LIN {X 0,Y 226.3,Z 547.719,A -85,B 0,C 180,E1 -21646.905,E2 -21646.905} C_VEL
LIN {X 0,Y 219.819,Z 558.471,A -85,B 0,C 180,E1 -21649.654,E2 -21649.654} C_VEL
LIN {X 0,Y 214.009,Z 567.653,A -85,B 0,C 180,E1 -21652.59,E2 -21652.59} C_VEL
LIN {X 0,Y 207.988,Z 576.689,A -85,B 0,C 180,E1 -21656.115,E2 -21656.115} C_VEL
LIN {X 0,Y 202.319,Z 585.085,A -85,B 0,C 180,E1 -21660.276,E2 -21660.276} C_VEL
LIN {X 0,Y 197.664,Z 592.031,A -85,B 0,C 180,E1 -21664.745,E2 -21664.745} C_VEL
LIN {X 0,Y 193.918,Z 597.973,A -85,B 0,C 180,E1 -21669.862,E2 -21669.862} C_VEL
LIN {X 0,Y 192.297,Z 600.784,A -85,B 0,C 180,E1 -21673,E2 -21673} C_VEL
LIN {X 0,Y 190.826,Z 603.573,A -85,B 0,C 180,E1 -21677.234,E2 -21677.234} C_VEL
LIN {X 0,Y 190.2,Z 605.482,A -85,B 0,C 180,E1 -21681.501,E2 -21681.501} C_VEL
LIN {X 0,Y 190.122,Z 606.399,A -85,B 0,C 180,E1 -21686.441,E2 -21686.441} C_VEL
LIN {X 0,Y 190.28,Z 606.307,A -85,B 0,C 180,E1 -21690.001,E2 -21690.001} C_VEL
LIN {X 0,Y 190.16,Z 605.178,A -85,B 0,C 180,E1 -21694.24,E2 -21694.24} C_VEL
LIN {X 0,Y 190.208,Z 603.116,A -85,B 0,C 180,E1 -21698.5,E2 -21698.5} C_VEL
LIN {X 0,Y 190.815,Z 599.908,A -85,B 0,C 180,E1 -21702.768,E2 -21702.768} C_VEL
LIN {X 0,Y 192.236,Z 595.672,A -85,B 0,C 180,E1 -21707.007,E2 -21707.007} C_VEL
LIN {X 0,Y 194.259,Z 590.216,A -85,B 0,C 180,E1 -21711.21,E2 -21711.21} C_VEL
LIN {X 0,Y 197.197,Z 583.475,A -85,B 0,C 180,E1 -21715.32,E2 -21715.32} C_VEL
LIN {X 0,Y 200.967,Z 575.348,A -85,B 0,C 180,E1 -21719.314,E2 -21719.314} C_VEL
LIN {X 0,Y 205.672,Z 565.618,A -85,B 0,C 180,E1 -21723.143,E2 -21723.143} C_VEL
LIN {X 0,Y 209.744,Z 557.011,A -85,B 0,C 180,E1 -21725.901,E2 -21725.901} C_VEL
LIN {X 0,Y 215.012,Z 545.421,A -85,B 0,C 180,E1 -21728.992,E2 -21728.992} C_VEL
LIN {X 0,Y 220.42,Z 532.769,A -85,B 0,C 180,E1 -21731.728,E2 -21731.728} C_VEL
LIN {X 0,Y 225.253,Z 520.818,A -85,B 0,C 180,E1 -21733.809,E2 -21733.809} C_VEL
LIN {X 0,Y 230.337,Z 506.753,A -85,B 0,C 180,E1 -21735.81,E2 -21735.81} C_VEL
LIN {X 0,Y 234.904,Z 492.399,A -85,B 0,C 180,E1 -21737.455,E2 -21737.455} C_VEL
LIN {X 0,Y 239.123,Z 476.927,A -85,B 0,C 180,E1 -21738.863,E2 -21738.863} C_VEL
LIN {X 0,Y 242.624,Z 461.116,A -85,B 0,C 180,E1 -21739.978,E2 -21739.978} C_VEL
LIN {X 0,Y 245.67,Z 444.06,A -85,B 0,C 180,E1 -21740.823,E2 -21740.823} C_VEL
LIN {X 0,Y 247.577,Z 427.936,A -85,B 0,C 180,E1 -21741.39,E2 -21741.39} C_VEL
LIN {X 0,Y 254.979,Z 326.261,A -85,B 0,C 180,E1 -21744.097,E2 -21744.097} C_VEL
LIN {X 0,Y 248.761,Z 313.085,A -85,B 0,C 180,E1 -21746.361,E2 -21746.361} C_VEL
LIN {X 0,Y 242.88,Z 301.521,A -85,B 0,C 180,E1 -21748.649,E2 -21748.649} C_VEL
LIN {X 0,Y 237.783,Z 292.318,A -85,B 0,C 180,E1 -21750.757,E2 -21750.757} C_VEL
LIN {X 0,Y 234.658,Z 287.086,A -85,B 0,C 180,E1 -21752.117,E2 -21752.117} C_VEL
LIN {X 0,Y 228.084,Z 277.705,A -85,B 0,C 180,E1 -21755.145,E2 -21755.145} C_VEL
LIN {X 0,Y 222.612,Z 270.114,A -85,B 0,C 180,E1 -21757.951,E2 -21757.951} C_VEL
LIN {X 0,Y 219.484,Z 266.04,A -85,B 0,C 180,E1 -21759.698,E2 -21759.698} C_VEL
LIN {X 0,Y 216.41,Z 261.942,A -85,B 0,C 180,E1 -21761.562,E2 -21761.562} C_VEL
LIN {X 0,Y 212.892,Z 257.748,A -85,B 0,C 180,E1 -21763.827,E2 -21763.827} C_VEL
LIN {X 0,Y 211.789,Z 256.222,A -85,B 0,C 180,E1 -21764.605,E2 -21764.605} C_VEL
LIN {X 0,Y 209.031,Z 253.204,A -85,B 0,C 180,E1 -21766.625,E2 -21766.625} C_VEL
LIN {X 0,Y 207.994,Z 251.231,A -85,B 0,C 180,E1 -21767.53,E2 -21767.53} C_VEL
LIN {X 0,Y 205.278,Z 248.973,A -85,B 0,C 180,E1 -21769.744,E2 -21769.744} C_VEL
LIN {X 0,Y 203.429,Z 245.607,A -85,B 0,C 180,E1 -21771.605,E2 -21771.605} C_VEL
LIN {X 0,Y 200.503,Z 243.62,A -85,B 0,C 180,E1 -21774.595,E2 -21774.595} C_VEL
LIN {X 0,Y 198.935,Z 241.093,A -85,B 0,C 180,E1 -21776.646,E2 -21776.646} C_VEL
LIN {X 0,Y 198.424,Z 239.663,A -85,B 0,C 180,E1 -21777.462,E2 -21777.462} C_VEL
LIN {X 0,Y 194.087,Z 236.776,A -85,B 0,C 180,E1 -21785.194,E2 -21785.194} C_VEL
LIN {X 0,Y 193.073,Z 234.315,A -85,B 0,C 180,E1 -21790.001,E2 -21790.001} C_VEL
LIN {X 0,Y 192.86,Z 234.123,A -85,B 0,C 180,E1 -21794.24,E2 -21794.24} C_VEL
LIN {X 0,Y 193.402,Z 236.089,A -85,B 0,C 180,E1 -21799.09,E2 -21799.09} C_VEL
LIN {X 0,Y 196.596,Z 239.298,A -85,B 0,C 180,E1 -21806.543,E2 -21806.543} C_VEL
LIN {X 0,Y 198.274,Z 240.054,A -85,B 0,C 180,E1 -21808.935,E2 -21808.935} C_VEL
LIN {X 0,Y 199.346,Z 242.603,A -85,B 0,C 180,E1 -21810.597,E2 -21810.597} C_VEL
LIN {X 0,Y 201.756,Z 245.019,A -85,B 0,C 180,E1 -21813.336,E2 -21813.336} C_VEL
LIN {X 0,Y 203.301,Z 246.022,A -85,B 0,C 180,E1 -21814.85,E2 -21814.85} C_VEL
LIN {X 0,Y 204.976,Z 248.974,A -85,B 0,C 180,E1 -21816.565,E2 -21816.565} C_VEL
LIN {X 0,Y 207.674,Z 251.22,A -85,B 0,C 180,E1 -21818.769,E2 -21818.769} C_VEL
LIN {X 0,Y 210.371,Z 255.153,A -85,B 0,C 180,E1 -21820.945,E2 -21820.945} C_VEL
LIN {X 0,Y 212.372,Z 257.041,A -85,B 0,C 180,E1 -21822.332,E2 -21822.332} C_VEL
LIN {X 0,Y 215.023,Z 260.684,A -85,B 0,C 180,E1 -21824.12,E2 -21824.12} C_VEL
LIN {X 0,Y 216.456,Z 262.166,A -85,B 0,C 180,E1 -21825.008,E2 -21825.008} C_VEL
LIN {X 0,Y 219.505,Z 266.13,A -85,B 0,C 180,E1 -21826.844,E2 -21826.844} C_VEL
LIN {X 0,Y 224.279,Z 272.472,A -85,B 0,C 180,E1 -21829.46,E2 -21829.46} C_VEL
LIN {X 0,Y 230.144,Z 280.518,A -85,B 0,C 180,E1 -21832.356,E2 -21832.356} C_VEL
LIN {X 0,Y 237.496,Z 291.276,A -85,B 0,C 180,E1 -21835.609,E2 -21835.609} C_VEL
LIN {X 0,Y 246.014,Z 305.014,A -85,B 0,C 180,E1 -21838.984,E2 -21838.984} C_VEL
LIN {X 0,Y 252.643,Z 316.674,A -85,B 0,C 180,E1 -21841.37,E2 -21841.37} C_VEL
LIN {X 0,Y 255.065,Z 321.147,A -85,B 0,C 180,E1 -21842.207,E2 -21842.207} C_VEL
LIN {X 0,Y 247.736,Z 420.872,A -85,B 0,C 180,E1 -21844.872,E2 -21844.872} C_VEL
LIN {X 0,Y 245.585,Z 437.685,A -85,B 0,C 180,E1 -21845.54,E2 -21845.54} C_VEL
LIN {X 0,Y 242.828,Z 453.469,A -85,B 0,C 180,E1 -21846.436,E2 -21846.436} C_VEL
LIN {X 0,Y 239.503,Z 468.656,A -85,B 0,C 180,E1 -21847.575,E2 -21847.575} C_VEL
LIN {X 0,Y 235.477,Z 483.687,A -85,B 0,C 180,E1 -21849.013,E2 -21849.013} C_VEL
LIN {X 0,Y 230.919,Z 498.153,A -85,B 0,C 180,E1 -21850.751,E2 -21850.751} C_VEL
LIN {X 0,Y 226.04,Z 511.98,A -85,B 0,C 180,E1 -21852.82,E2 -21852.82} C_VEL
LIN {X 0,Y 220.734,Z 525.239,A -85,B 0,C 180,E1 -21855.243,E2 -21855.243} C_VEL
LIN {X 0,Y 215.258,Z 537.956,A -85,B 0,C 180,E1 -21858.134,E2 -21858.134} C_VEL
LIN {X 0,Y 209.942,Z 549.371,A -85,B 0,C 180,E1 -21861.335,E2 -21861.335} C_VEL
LIN {X 0,Y 205.245,Z 559.035,A -85,B 0,C 180,E1 -21864.704,E2 -21864.704} C_VEL
LIN {X 0,Y 200.912,Z 567.881,A -85,B 0,C 180,E1 -21868.496,E2 -21868.496} C_VEL
LIN {X 0,Y 197.029,Z 575.994,A -85,B 0,C 180,E1 -21872.859,E2 -21872.859} C_VEL
LIN {X 0,Y 194.041,Z 582.465,A -85,B 0,C 180,E1 -21877.282,E2 -21877.282} C_VEL
LIN {X 0,Y 192.072,Z 587.326,A -85,B 0,C 180,E1 -21881.609,E2 -21881.609} C_VEL
LIN {X 0,Y 190.587,Z 591.369,A -85,B 0,C 180,E1 -21886.512,E2 -21886.512} C_VEL
LIN {X 0,Y 189.824,Z 594.152,A -85,B 0,C 180,E1 -21891.729,E2 -21891.729} C_VEL
LIN {X 0,Y 189.656,Z 595.421,A -85,B 0,C 180,E1 -21896.402,E2 -21896.402} C_VEL
LIN {X 0,Y 189.956,Z 595.502,A -85,B 0,C 180,E1 -21901.195,E2 -21901.195} C_VEL
LIN {X 0,Y 190.879,Z 594.328,A -85,B 0,C 180,E1 -21906.092,E2 -21906.092} C_VEL
LIN {X 0,Y 192.629,Z 591.858,A -85,B 0,C 180,E1 -21911.049,E2 -21911.049} C_VEL
LIN {X 0,Y 195.361,Z 587.97,A -85,B 0,C 180,E1 -21916.011,E2 -21916.011} C_VEL
LIN {X 0,Y 199.252,Z 582.546,A -85,B 0,C 180,E1 -21920.892,E2 -21920.892} C_VEL
LIN {X 0,Y 203.207,Z 577.04,A -85,B 0,C 180,E1 -21924.614,E2 -21924.614} C_VEL
LIN {X 0,Y 209.079,Z 568.863,A -85,B 0,C 180,E1 -21928.937,E2 -21928.937} C_VEL
LIN {X 0,Y 214.504,Z 561.069,A -85,B 0,C 180,E1 -21932.203,E2 -21932.203} C_VEL
LIN {X 0,Y 221.257,Z 550.841,A -85,B 0,C 180,E1 -21935.611,E2 -21935.611} C_VEL
LIN {X 0,Y 228.118,Z 539.48,A -85,B 0,C 180,E1 -21938.616,E2 -21938.616} C_VEL
LIN {X 0,Y 234.856,Z 527.408,A -85,B 0,C 180,E1 -21941.148,E2 -21941.148} C_VEL
LIN {X 0,Y 241.301,Z 514.567,A -85,B 0,C 180,E1 -21943.339,E2 -21943.339} C_VEL
LIN {X 0,Y 247.296,Z 501.19,A -85,B 0,C 180,E1 -21945.181,E2 -21945.181} C_VEL
LIN {X 0,Y 252.741,Z 487.284,A -85,B 0,C 180,E1 -21946.713,E2 -21946.713} C_VEL
LIN {X 0,Y 257.863,Z 471.68,A -85,B 0,C 180,E1 -21948.089,E2 -21948.089} C_VEL
LIN {X 0,Y 261.833,Z 457.05,A -85,B 0,C 180,E1 -21949.095,E2 -21949.095} C_VEL
LIN {X 0,Y 265.125,Z 441.997,A -85,B 0,C 180,E1 -21949.899,E2 -21949.899} C_VEL
LIN {X 0,Y 267.848,Z 425.319,A -85,B 0,C 180,E1 -21950.519,E2 -21950.519} C_VEL
LIN {X 0,Y 272.094,Z 380.522,A -85,B 0,C 180,E1 -21951.669,E2 -21951.669} C_VEL
LIN {X 0,Y 276.451,Z 332.828,A -85,B 0,C 180,E1 -21952.851,E2 -21952.851} C_VEL
LIN {X 0,Y 272.688,Z 325.115,A -85,B 0,C 180,E1 -21955.176,E2 -21955.176} C_VEL
LIN {X 0,Y 268.508,Z 317.322,A -85,B 0,C 180,E1 -21958.203,E2 -21958.203} C_VEL
LIN {X 0,Y 266.207,Z 313.483,A -85,B 0,C 180,E1 -21960.156,E2 -21960.156} C_VEL
LIN {X 0,Y 263.602,Z 308.901,A -85,B 0,C 180,E1 -21962.925,E2 -21962.925} C_VEL
LIN {X 0,Y 262.122,Z 306.157,A -85,B 0,C 180,E1 -21964.992,E2 -21964.992} C_VEL
LIN {X 0,Y 260.235,Z 303.911,A -85,B 0,C 180,E1 -21968.582,E2 -21968.582} C_VEL
LIN {X 0,Y 259.761,Z 301.619,A -85,B 0,C 180,E1 -21971.359,E2 -21971.359} C_VEL
LIN {X 0,Y 259.671,Z 301.612,A -85,B 0,C 180,E1 -21973.484,E2 -21973.484} C_VEL
LIN {X 0,Y 261.393,Z 305.792,A -85,B 0,C 180,E1 -21979.607,E2 -21979.607} C_VEL
LIN {X 0,Y 261.99,Z 306.539,A -85,B 0,C 180,E1 -21980.538,E2 -21980.538} C_VEL
LIN {X 0,Y 263.625,Z 309.473,A -85,B 0,C 180,E1 -21982.8,E2 -21982.8} C_VEL
LIN {X 0,Y 264.588,Z 311.792,A -85,B 0,C 180,E1 -21983.958,E2 -21983.958} C_VEL
LIN {X 0,Y 265.403,Z 315.135,A -85,B 0,C 180,E1 -21985.005,E2 -21985.005} C_VEL
LIN {X 0,Y 266.944,Z 323.106,A -85,B 0,C 180,E1 -21986.933,E2 -21986.933} C_VEL
LIN {X 0,Y 268.315,Z 328.069,A -85,B 0,C 180,E1 -21988.267,E2 -21988.267} C_VEL
LIN {X 0,Y 270.696,Z 333.766,A -85,B 0,C 180,E1 -21990.065,E2 -21990.065} C_VEL
LIN {X 0,Y 272.946,Z 339.745,A -85,B 0,C 180,E1 -21991.648,E2 -21991.648} C_VEL
LIN {X 0,Y 264.303,Z 430.241,A -85,B 0,C 180,E1 -21993.891,E2 -21993.891} C_VEL
LIN {X 0,Y 261.773,Z 445.91,A -85,B 0,C 180,E1 -21994.435,E2 -21994.435} C_VEL
LIN {X 0,Y 257.966,Z 462.562,A -85,B 0,C 180,E1 -21995.185,E2 -21995.185} C_VEL
LIN {X 0,Y 253.496,Z 478.126,A -85,B 0,C 180,E1 -21996.152,E2 -21996.152} C_VEL
LIN {X 0,Y 247.91,Z 494.137,A -85,B 0,C 180,E1 -21997.462,E2 -21997.462} C_VEL
LIN {X 0,Y 241.934,Z 508.77,A -85,B 0,C 180,E1 -21999.009,E2 -21999.009} C_VEL
LIN {X 0,Y 235.575,Z 522.278,A -85,B 0,C 180,E1 -22000.799,E2 -22000.799} C_VEL
LIN {X 0,Y 229.471,Z 533.923,A -85,B 0,C 180,E1 -22002.69,E2 -22002.69} C_VEL
LIN {X 0,Y 222.174,Z 546.633,A -85,B 0,C 180,E1 -22005.266,E2 -22005.266} C_VEL
LIN {X 0,Y 214.44,Z 558.899,A -85,B 0,C 180,E1 -22008.421,E2 -22008.421} C_VEL
LIN {X 0,Y 207.554,Z 569.21,A -85,B 0,C 180,E1 -22011.834,E2 -22011.834} C_VEL
LIN {X 0,Y 201.341,Z 577.918,A -85,B 0,C 180,E1 -22015.444,E2 -22015.444} C_VEL
LIN {X 0,Y 195.442,Z 586.085,A -85,B 0,C 180,E1 -22019.774,E2 -22019.774} C_VEL
LIN {X 0,Y 191.179,Z 592.098,A -85,B 0,C 180,E1 -22023.825,E2 -22023.825} C_VEL
LIN {X 0,Y 187.164,Z 597.975,A -85,B 0,C 180,E1 -22029.102,E2 -22029.102} C_VEL
LIN {X 0,Y 184.556,Z 602.217,A -85,B 0,C 180,E1 -22034.541,E2 -22034.541} C_VEL
LIN {X 0,Y 183.396,Z 604.501,A -85,B 0,C 180,E1 -22038.954,E2 -22038.954} C_VEL
LIN {X 0,Y 182.995,Z 605.853,A -85,B 0,C 180,E1 -22043.385,E2 -22043.385} C_VEL
LIN {X 0,Y 183.056,Z 606.213,A -85,B 0,C 180,E1 -22047.8,E2 -22047.8} C_VEL
LIN {X 0,Y 183.184,Z 606.069,A -85,B 0,C 180,E1 -22050.001,E2 -22050.001} C_VEL
LIN {X 0,Y 183.072,Z 604.899,A -85,B 0,C 180,E1 -22054.404,E2 -22054.404} C_VEL
LIN {X 0,Y 183.146,Z 602.78,A -85,B 0,C 180,E1 -22058.83,E2 -22058.83} C_VEL
LIN {X 0,Y 184.161,Z 598.607,A -85,B 0,C 180,E1 -22064.363,E2 -22064.363} C_VEL
LIN {X 0,Y 186.011,Z 593.473,A -85,B 0,C 180,E1 -22069.167,E2 -22069.167} C_VEL
LIN {X 0,Y 188.244,Z 588.146,A -85,B 0,C 180,E1 -22073.08,E2 -22073.08} C_VEL
LIN {X 0,Y 191.587,Z 581.058,A -85,B 0,C 180,E1 -22077.293,E2 -22077.293} C_VEL
LIN {X 0,Y 195.858,Z 572.422,A -85,B 0,C 180,E1 -22081.353,E2 -22081.353} C_VEL
LIN {X 0,Y 200.377,Z 563.506,A -85,B 0,C 180,E1 -22084.747,E2 -22084.747} C_VEL
LIN {X 0,Y 205.384,Z 553.105,A -85,B 0,C 180,E1 -22088.02,E2 -22088.02} C_VEL
LIN {X 0,Y 211.125,Z 540.871,A -85,B 0,C 180,E1 -22091.105,E2 -22091.105} C_VEL
LIN {X 0,Y 216.562,Z 528.481,A -85,B 0,C 180,E1 -22093.6,E2 -22093.6} C_VEL
LIN {X 0,Y 221.922,Z 514.889,A -85,B 0,C 180,E1 -22095.836,E2 -22095.836} C_VEL
LIN {X 0,Y 226.912,Z 500.869,A -85,B 0,C 180,E1 -22097.686,E2 -22097.686} C_VEL
LIN {X 0,Y 231.705,Z 485.342,A -85,B 0,C 180,E1 -22099.314,E2 -22099.314} C_VEL
LIN {X 0,Y 235.829,Z 469.309,A -85,B 0,C 180,E1 -22100.621,E2 -22100.621} C_VEL
LIN {X 0,Y 239.096,Z 453.413,A -85,B 0,C 180,E1 -22101.585,E2 -22101.585} C_VEL
LIN {X 0,Y 241.685,Z 437.265,A -85,B 0,C 180,E1 -22102.272,E2 -22102.272} C_VEL
LIN {X 0,Y 243.531,Z 417.107,A -85,B 0,C 180,E1 -22102.898,E2 -22102.898} C_VEL
LIN {X 0,Y 250.181,Z 328.977,A -85,B 0,C 180,E1 -22105.231,E2 -22105.231} C_VEL
LIN {X 0,Y 243.246,Z 314.287,A -85,B 0,C 180,E1 -22107.888,E2 -22107.888} C_VEL
LIN {X 0,Y 236.492,Z 301.128,A -85,B 0,C 180,E1 -22110.706,E2 -22110.706} C_VEL
LIN {X 0,Y 231.829,Z 292.97,A -85,B 0,C 180,E1 -22112.792,E2 -22112.792} C_VEL
LIN {X 0,Y 224.763,Z 282.709,A -85,B 0,C 180,E1 -22116.179,E2 -22116.179} C_VEL
LIN {X 0,Y 219.991,Z 276.007,A -85,B 0,C 180,E1 -22118.737,E2 -22118.737} C_VEL
LIN {X 0,Y 216.99,Z 272.049,A -85,B 0,C 180,E1 -22120.48,E2 -22120.48} C_VEL
LIN {X 0,Y 213.383,Z 267.331,A -85,B 0,C 180,E1 -22122.757,E2 -22122.757} C_VEL
LIN {X 0,Y 210.463,Z 263.477,A -85,B 0,C 180,E1 -22124.764,E2 -22124.764} C_VEL
LIN {X 0,Y 206.967,Z 259.331,A -85,B 0,C 180,E1 -22127.435,E2 -22127.435} C_VEL
LIN {X 0,Y 205.872,Z 257.674,A -85,B 0,C 180,E1 -22128.38,E2 -22128.38} C_VEL
LIN {X 0,Y 203.302,Z 255.168,A -85,B 0,C 180,E1 -22130.597,E2 -22130.597} C_VEL
LIN {X 0,Y 201.743,Z 252.369,A -85,B 0,C 180,E1 -22132.242,E2 -22132.242} C_VEL
LIN {X 0,Y 198.832,Z 250.084,A -85,B 0,C 180,E1 -22135.391,E2 -22135.391} C_VEL
LIN {X 0,Y 197.37,Z 247.437,A -85,B 0,C 180,E1 -22137.441,E2 -22137.441} C_VEL
LIN {X 0,Y 197.068,Z 246.554,A -85,B 0,C 180,E1 -22137.956,E2 -22137.956} C_VEL
LIN {X 0,Y 192.948,Z 243.573,A -85,B 0,C 180,E1 -22145.749,E2 -22145.749} C_VEL
LIN {X 0,Y 192.092,Z 241.306,A -85,B 0,C 180,E1 -22150.235,E2 -22150.235} C_VEL
LIN {X 0,Y 191.895,Z 241.115,A -85,B 0,C 180,E1 -22153.772,E2 -22153.772} C_VEL
LIN {X 0,Y 192.338,Z 242.935,A -85,B 0,C 180,E1 -22158.591,E2 -22158.591} C_VEL
LIN {X 0,Y 195.167,Z 246.109,A -85,B 0,C 180,E1 -22165.809,E2 -22165.809} C_VEL
LIN {X 0,Y 196.89,Z 246.955,A -85,B 0,C 180,E1 -22168.377,E2 -22168.377} C_VEL
LIN {X 0,Y 198.457,Z 250.027,A -85,B 0,C 180,E1 -22170.749,E2 -22170.749} C_VEL
LIN {X 0,Y 201.129,Z 252.313,A -85,B 0,C 180,E1 -22173.699,E2 -22173.699} C_VEL
LIN {X 0,Y 201.816,Z 253.005,A -85,B 0,C 180,E1 -22174.409,E2 -22174.409} C_VEL
LIN {X 0,Y 203.854,Z 256.203,A -85,B 0,C 180,E1 -22176.491,E2 -22176.491} C_VEL
LIN {X 0,Y 206.224,Z 258.311,A -85,B 0,C 180,E1 -22178.474,E2 -22178.474} C_VEL
LIN {X 0,Y 208.536,Z 261.69,A -85,B 0,C 180,E1 -22180.376,E2 -22180.376} C_VEL
LIN {X 0,Y 210.45,Z 263.668,A -85,B 0,C 180,E1 -22181.764,E2 -22181.764} C_VEL
LIN {X 0,Y 213.581,Z 267.699,A -85,B 0,C 180,E1 -22183.906,E2 -22183.906} C_VEL
LIN {X 0,Y 218.451,Z 274.056,A -85,B 0,C 180,E1 -22186.916,E2 -22186.916} C_VEL
LIN {X 0,Y 223.976,Z 281.525,A -85,B 0,C 180,E1 -22189.934,E2 -22189.934} C_VEL
LIN {X 0,Y 231.139,Z 291.963,A -85,B 0,C 180,E1 -22193.409,E2 -22193.409} C_VEL
LIN {X 0,Y 237.448,Z 301.854,A -85,B 0,C 180,E1 -22196.169,E2 -22196.169} C_VEL
LIN {X 0,Y 245.36,Z 315.183,A -85,B 0,C 180,E1 -22199.295,E2 -22199.295} C_VEL
LIN {X 0,Y 250.208,Z 324.114,A -85,B 0,C 180,E1 -22201.067,E2 -22201.067} C_VEL
LIN {X 0,Y 242.664,Z 422.976,A -85,B 0,C 180,E1 -22203.731,E2 -22203.731} C_VEL
LIN {X 0,Y 240.324,Z 440,A -85,B 0,C 180,E1 -22204.447,E2 -22204.447} C_VEL
LIN {X 0,Y 237.325,Z 455.867,A -85,B 0,C 180,E1 -22205.39,E2 -22205.39} C_VEL
LIN {X 0,Y 233.921,Z 470.539,A -85,B 0,C 180,E1 -22206.541,E2 -22206.541} C_VEL
LIN {X 0,Y 229.831,Z 485.302,A -85,B 0,C 180,E1 -22208.001,E2 -22208.001} C_VEL
LIN {X 0,Y 224.788,Z 500.514,A -85,B 0,C 180,E1 -22209.884,E2 -22209.884} C_VEL
LIN {X 0,Y 219.617,Z 514.379,A -85,B 0,C 180,E1 -22212.06,E2 -22212.06} C_VEL
LIN {X 0,Y 214.603,Z 526.286,A -85,B 0,C 180,E1 -22214.325,E2 -22214.325} C_VEL
LIN {X 0,Y 208.931,Z 538.914,A -85,B 0,C 180,E1 -22217.29,E2 -22217.29} C_VEL
LIN {X 0,Y 203.471,Z 550.176,A -85,B 0,C 180,E1 -22220.556,E2 -22220.556} C_VEL
LIN {X 0,Y 198.74,Z 559.505,A -85,B 0,C 180,E1 -22223.91,E2 -22223.91} C_VEL
LIN {X 0,Y 194.114,Z 568.532,A -85,B 0,C 180,E1 -22227.925,E2 -22227.925} C_VEL
LIN {X 0,Y 190.362,Z 576.056,A -85,B 0,C 180,E1 -22232.115,E2 -22232.115} C_VEL
LIN {X 0,Y 187.322,Z 582.298,A -85,B 0,C 180,E1 -22236.462,E2 -22236.462} C_VEL
LIN {X 0,Y 185.204,Z 587.21,A -85,B 0,C 180,E1 -22240.937,E2 -22240.937} C_VEL
LIN {X 0,Y 183.694,Z 591.029,A -85,B 0,C 180,E1 -22245.533,E2 -22245.533} C_VEL
LIN {X 0,Y 182.822,Z 593.775,A -85,B 0,C 180,E1 -22250.24,E2 -22250.24} C_VEL
LIN {X 0,Y 182.536,Z 595.332,A -85,B 0,C 180,E1 -22255.056,E2 -22255.056} C_VEL
LIN {X 0,Y 182.588,Z 595.725,A -85,B 0,C 180,E1 -22257.713,E2 -22257.713} C_VEL
LIN {X 0,Y 183.027,Z 595.601,A -85,B 0,C 180,E1 -22262.518,E2 -22262.518} C_VEL
LIN {X 0,Y 184.195,Z 594.221,A -85,B 0,C 180,E1 -22267.623,E2 -22267.623} C_VEL
LIN {X 0,Y 186.313,Z 591.474,A -85,B 0,C 180,E1 -22272.763,E2 -22272.763} C_VEL
LIN {X 0,Y 189.494,Z 587.299,A -85,B 0,C 180,E1 -22277.88,E2 -22277.88} C_VEL
LIN {X 0,Y 193.89,Z 581.559,A -85,B 0,C 180,E1 -22282.884,E2 -22282.884} C_VEL
LIN {X 0,Y 198.881,Z 575.19,A -85,B 0,C 180,E1 -22287.061,E2 -22287.061} C_VEL
LIN {X 0,Y 204.17,Z 568.171,A -85,B 0,C 180,E1 -22290.654,E2 -22290.654} C_VEL
LIN {X 0,Y 210.637,Z 559.222,A -85,B 0,C 180,E1 -22294.294,E2 -22294.294} C_VEL
LIN {X 0,Y 217.462,Z 549.157,A -85,B 0,C 180,E1 -22297.542,E2 -22297.542} C_VEL
LIN {X 0,Y 224.655,Z 537.774,A -85,B 0,C 180,E1 -22300.457,E2 -22300.457} C_VEL
LIN {X 0,Y 232.036,Z 524.859,A -85,B 0,C 180,E1 -22303.08,E2 -22303.08} C_VEL
LIN {X 0,Y 239.031,Z 510.982,A -85,B 0,C 180,E1 -22305.316,E2 -22305.316} C_VEL
LIN {X 0,Y 245.137,Z 497.106,A -85,B 0,C 180,E1 -22307.096,E2 -22307.096} C_VEL
LIN {X 0,Y 250.914,Z 482.098,A -85,B 0,C 180,E1 -22308.613,E2 -22308.613} C_VEL
LIN {X 0,Y 256.012,Z 466.15,A -85,B 0,C 180,E1 -22309.889,E2 -22309.889} C_VEL
LIN {X 0,Y 259.969,Z 450.749,A -85,B 0,C 180,E1 -22310.852,E2 -22310.852} C_VEL
LIN {X 0,Y 263.326,Z 433.993,A -85,B 0,C 180,E1 -22311.595,E2 -22311.595} C_VEL
LIN {X 0,Y 265.649,Z 416.43,A -85,B 0,C 180,E1 -22312.131,E2 -22312.131} C_VEL
LIN {X 0,Y 273.16,Z 336.704,A -85,B 0,C 180,E1 -22314.093,E2 -22314.093} C_VEL
LIN {X 0,Y 269.895,Z 329.796,A -85,B 0,C 180,E1 -22316.306,E2 -22316.306} C_VEL
LIN {X 0,Y 266.062,Z 322.464,A -85,B 0,C 180,E1 -22319.353,E2 -22319.353} C_VEL
LIN {X 0,Y 264.364,Z 319.548,A -85,B 0,C 180,E1 -22320.947,E2 -22320.947} C_VEL
LIN {X 0,Y 262.224,Z 315.543,A -85,B 0,C 180,E1 -22323.392,E2 -22323.392} C_VEL
LIN {X 0,Y 261.069,Z 313.166,A -85,B 0,C 180,E1 -22325.114,E2 -22325.114} C_VEL
LIN {X 0,Y 259.172,Z 310.79,A -85,B 0,C 180,E1 -22328.901,E2 -22328.901} C_VEL
LIN {X 0,Y 258.767,Z 308.505,A -85,B 0,C 180,E1 -22331.875,E2 -22331.875} C_VEL
LIN {X 0,Y 258.727,Z 308.886,A -85,B 0,C 180,E1 -22333.842,E2 -22333.842} C_VEL
LIN {X 0,Y 260.193,Z 312.651,A -85,B 0,C 180,E1 -22339.219,E2 -22339.219} C_VEL
LIN {X 0,Y 260.816,Z 313.445,A -85,B 0,C 180,E1 -22340.238,E2 -22340.238} C_VEL
LIN {X 0,Y 263.23,Z 317.763,A -85,B 0,C 180,E1 -22343.494,E2 -22343.494} C_VEL
LIN {X 0,Y 265.72,Z 322.247,A -85,B 0,C 180,E1 -22346.012,E2 -22346.012} C_VEL
LIN {X 0,Y 268.315,Z 328.069,A -85,B 0,C 180,E1 -22348.267,E2 -22348.267} C_VEL
LIN {X 0,Y 269.259,Z 331.681,A -85,B 0,C 180,E1 -22349.117,E2 -22349.117} C_VEL
LIN {X 0,Y 269.791,Z 336.203,A -85,B 0,C 180,E1 -22349.768,E2 -22349.768} C_VEL
LIN {X 0,Y 269.902,Z 341.303,A -85,B 0,C 180,E1 -22350.22,E2 -22350.22} C_VEL
LIN {X 0,Y 269.552,Z 346.705,A -85,B 0,C 180,E1 -22350.448,E2 -22350.448} C_VEL
LIN {X 0,Y 261.1,Z 431.121,A -85,B 0,C 180,E1 -22352.522,E2 -22352.522} C_VEL
LIN {X 0,Y 258.109,Z 448.401,A -85,B 0,C 180,E1 -22353.125,E2 -22353.125} C_VEL
LIN {X 0,Y 254.028,Z 465.034,A -85,B 0,C 180,E1 -22353.905,E2 -22353.905} C_VEL
LIN {X 0,Y 249.452,Z 479.983,A -85,B 0,C 180,E1 -22354.861,E2 -22354.861} C_VEL
LIN {X 0,Y 243.746,Z 495.578,A -85,B 0,C 180,E1 -22356.166,E2 -22356.166} C_VEL
LIN {X 0,Y 237.589,Z 509.95,A -85,B 0,C 180,E1 -22357.697,E2 -22357.697} C_VEL
LIN {X 0,Y 230.46,Z 524.354,A -85,B 0,C 180,E1 -22359.647,E2 -22359.647} C_VEL
LIN {X 0,Y 222.573,Z 538.485,A -85,B 0,C 180,E1 -22362.096,E2 -22362.096} C_VEL
LIN {X 0,Y 215.102,Z 550.426,A -85,B 0,C 180,E1 -22364.715,E2 -22364.715} C_VEL
LIN {X 0,Y 208.22,Z 560.671,A -85,B 0,C 180,E1 -22367.543,E2 -22367.543} C_VEL
LIN {X 0,Y 201.985,Z 569.544,A -85,B 0,C 180,E1 -22370.581,E2 -22370.581} C_VEL
LIN {X 0,Y 195.486,Z 578.155,A -85,B 0,C 180,E1 -22374.254,E2 -22374.254} C_VEL
LIN {X 0,Y 189.266,Z 586.23,A -85,B 0,C 180,E1 -22378.678,E2 -22378.678} C_VEL
LIN {X 0,Y 184.755,Z 592.149,A -85,B 0,C 180,E1 -22382.841,E2 -22382.841} C_VEL
LIN {X 0,Y 181.22,Z 596.894,A -85,B 0,C 180,E1 -22387.182,E2 -22387.182} C_VEL
LIN {X 0,Y 178.621,Z 600.654,A -85,B 0,C 180,E1 -22391.654,E2 -22391.654} C_VEL
LIN {X 0,Y 176.858,Z 603.368,A -85,B 0,C 180,E1 -22396.207,E2 -22396.207} C_VEL
LIN {X 0,Y 176.066,Z 605.159,A -85,B 0,C 180,E1 -22400.813,E2 -22400.813} C_VEL
LIN {X 0,Y 175.933,Z 605.949,A -85,B 0,C 180,E1 -22405.418,E2 -22405.418} C_VEL
LIN {X 0,Y 176.09,Z 605.819,A -85,B 0,C 180,E1 -22410.001,E2 -22410.001} C_VEL
LIN {X 0,Y 175.966,Z 604.619,A -85,B 0,C 180,E1 -22414.582,E2 -22414.582} C_VEL
LIN {X 0,Y 176.07,Z 602.438,A -85,B 0,C 180,E1 -22419.188,E2 -22419.188} C_VEL
LIN {X 0,Y 176.85,Z 599.162,A -85,B 0,C 180,E1 -22423.795,E2 -22423.795} C_VEL
LIN {X 0,Y 178.51,Z 594.789,A -85,B 0,C 180,E1 -22428.359,E2 -22428.359} C_VEL
LIN {X 0,Y 180.873,Z 589.259,A -85,B 0,C 180,E1 -22432.865,E2 -22432.865} C_VEL
LIN {X 0,Y 184.22,Z 582.367,A -85,B 0,C 180,E1 -22437.246,E2 -22437.246} C_VEL
LIN {X 0,Y 188.477,Z 574.073,A -85,B 0,C 180,E1 -22441.469,E2 -22441.469} C_VEL
LIN {X 0,Y 193.023,Z 565.54,A -85,B 0,C 180,E1 -22444.992,E2 -22444.992} C_VEL
LIN {X 0,Y 198.074,Z 555.637,A -85,B 0,C 180,E1 -22448.302,E2 -22448.302} C_VEL
LIN {X 0,Y 203.947,Z 543.609,A -85,B 0,C 180,E1 -22451.556,E2 -22451.556} C_VEL
LIN {X 0,Y 209.412,Z 531.767,A -85,B 0,C 180,E1 -22454.138,E2 -22454.138} C_VEL
LIN {X 0,Y 215.029,Z 518.632,A -85,B 0,C 180,E1 -22456.453,E2 -22456.453} C_VEL
LIN {X 0,Y 220.495,Z 504.06,A -85,B 0,C 180,E1 -22458.507,E2 -22458.507} C_VEL
LIN {X 0,Y 225.408,Z 489.172,A -85,B 0,C 180,E1 -22460.155,E2 -22460.155} C_VEL
LIN {X 0,Y 229.609,Z 474.055,A -85,B 0,C 180,E1 -22461.484,E2 -22461.484} C_VEL
LIN {X 0,Y 233.053,Z 459.032,A -85,B 0,C 180,E1 -22462.512,E2 -22462.512} C_VEL
LIN {X 0,Y 236.22,Z 441.561,A -85,B 0,C 180,E1 -22463.357,E2 -22463.357} C_VEL
LIN {X 0,Y 237.982,Z 426.238,A -85,B 0,C 180,E1 -22463.885,E2 -22463.885} C_VEL
LIN {X 0,Y 245.348,Z 331.649,A -85,B 0,C 180,E1 -22466.42,E2 -22466.42} C_VEL
LIN {X 0,Y 239.237,Z 318.455,A -85,B 0,C 180,E1 -22468.904,E2 -22468.904} C_VEL
LIN {X 0,Y 233.163,Z 306.362,A -85,B 0,C 180,E1 -22471.547,E2 -22471.547} C_VEL
LIN {X 0,Y 228.758,Z 298.512,A -85,B 0,C 180,E1 -22473.608,E2 -22473.608} C_VEL
LIN {X 0,Y 222.146,Z 288.693,A -85,B 0,C 180,E1 -22476.9,E2 -22476.9} C_VEL
LIN {X 0,Y 217.153,Z 281.57,A -85,B 0,C 180,E1 -22479.687,E2 -22479.687} C_VEL
LIN {X 0,Y 214.613,Z 278.145,A -85,B 0,C 180,E1 -22481.23,E2 -22481.23} C_VEL
LIN {X 0,Y 211.048,Z 273.421,A -85,B 0,C 180,E1 -22483.558,E2 -22483.558} C_VEL
LIN {X 0,Y 207.766,Z 269.077,A -85,B 0,C 180,E1 -22485.945,E2 -22485.945} C_VEL
LIN {X 0,Y 204.958,Z 265.496,A -85,B 0,C 180,E1 -22488.228,E2 -22488.228} C_VEL
LIN {X 0,Y 204.025,Z 264.217,A -85,B 0,C 180,E1 -22489.041,E2 -22489.041} C_VEL
LIN {X 0,Y 201.541,Z 261.585,A -85,B 0,C 180,E1 -22491.297,E2 -22491.297} C_VEL
LIN {X 0,Y 200.167,Z 259.106,A -85,B 0,C 180,E1 -22492.815,E2 -22492.815} C_VEL
LIN {X 0,Y 197.499,Z 256.908,A -85,B 0,C 180,E1 -22495.807,E2 -22495.807} C_VEL
LIN {X 0,Y 195.908,Z 253.963,A -85,B 0,C 180,E1 -22498.134,E2 -22498.134} C_VEL
LIN {X 0,Y 195.494,Z 253.311,A -85,B 0,C 180,E1 -22498.791,E2 -22498.791} C_VEL
LIN {X 0,Y 191.881,Z 250.487,A -85,B 0,C 180,E1 -22506.111,E2 -22506.111} C_VEL
LIN {X 0,Y 191.101,Z 248.253,A -85,B 0,C 180,E1 -22510.596,E2 -22510.596} C_VEL
LIN {X 0,Y 190.945,Z 248.21,A -85,B 0,C 180,E1 -22513.842,E2 -22513.842} C_VEL
LIN {X 0,Y 191.355,Z 249.955,A -85,B 0,C 180,E1 -22518.448,E2 -22518.448} C_VEL
LIN {X 0,Y 194.165,Z 253.137,A -85,B 0,C 180,E1 -22525.744,E2 -22525.744} C_VEL
LIN {X 0,Y 195.596,Z 253.892,A -85,B 0,C 180,E1 -22527.938,E2 -22527.938} C_VEL
LIN {X 0,Y 197.167,Z 256.919,A -85,B 0,C 180,E1 -22530.379,E2 -22530.379} C_VEL
LIN {X 0,Y 200.233,Z 259.722,A -85,B 0,C 180,E1 -22533.833,E2 -22533.833} C_VEL
LIN {X 0,Y 202.464,Z 263.095,A -85,B 0,C 180,E1 -22536.165,E2 -22536.165} C_VEL
LIN {X 0,Y 204.485,Z 265.008,A -85,B 0,C 180,E1 -22537.92,E2 -22537.92} C_VEL
LIN {X 0,Y 207.16,Z 268.673,A -85,B 0,C 180,E1 -22540.134,E2 -22540.134} C_VEL
LIN {X 0,Y 208.52,Z 270.206,A -85,B 0,C 180,E1 -22541.161,E2 -22541.161} C_VEL
LIN {X 0,Y 211.842,Z 274.414,A -85,B 0,C 180,E1 -22543.498,E2 -22543.498} C_VEL
LIN {X 0,Y 215.316,Z 279.011,A -85,B 0,C 180,E1 -22545.729,E2 -22545.729} C_VEL
LIN {X 0,Y 221.715,Z 288.042,A -85,B 0,C 180,E1 -22549.39,E2 -22549.39} C_VEL
LIN {X 0,Y 228.614,Z 298.283,A -85,B 0,C 180,E1 -22552.847,E2 -22552.847} C_VEL
LIN {X 0,Y 235.272,Z 309.039,A -85,B 0,C 180,E1 -22555.84,E2 -22555.84} C_VEL
LIN {X 0,Y 243.156,Z 322.747,A -85,B 0,C 180,E1 -22559.025,E2 -22559.025} C_VEL
LIN {X 0,Y 245.392,Z 327.043,A -85,B 0,C 180,E1 -22559.883,E2 -22559.883} C_VEL
LIN {X 0,Y 239.598,Z 402.31,A -85,B 0,C 180,E1 -22561.9,E2 -22561.9} C_VEL
LIN {X 0,Y 237.462,Z 425.785,A -85,B 0,C 180,E1 -22562.586,E2 -22562.586} C_VEL
LIN {X 0,Y 235.001,Z 442.694,A -85,B 0,C 180,E1 -22563.346,E2 -22563.346} C_VEL
LIN {X 0,Y 231.645,Z 459.326,A -85,B 0,C 180,E1 -22564.384,E2 -22564.384} C_VEL
LIN {X 0,Y 227.356,Z 476.259,A -85,B 0,C 180,E1 -22565.821,E2 -22565.821} C_VEL
LIN {X 0,Y 222.667,Z 491.538,A -85,B 0,C 180,E1 -22567.499,E2 -22567.499} C_VEL
LIN {X 0,Y 217.868,Z 504.887,A -85,B 0,C 180,E1 -22569.306,E2 -22569.306} C_VEL
LIN {X 0,Y 212.271,Z 518.894,A -85,B 0,C 180,E1 -22571.667,E2 -22571.667} C_VEL
LIN {X 0,Y 206.784,Z 531.223,A -85,B 0,C 180,E1 -22574.222,E2 -22574.222} C_VEL
LIN {X 0,Y 200.823,Z 543.657,A -85,B 0,C 180,E1 -22577.445,E2 -22577.445} C_VEL
LIN {X 0,Y 195.584,Z 553.744,A -85,B 0,C 180,E1 -22580.694,E2 -22580.694} C_VEL
LIN {X 0,Y 190.69,Z 562.923,A -85,B 0,C 180,E1 -22584.324,E2 -22584.324} C_VEL
LIN {X 0,Y 186.827,Z 570.22,A -85,B 0,C 180,E1 -22587.844,E2 -22587.844} C_VEL
LIN {X 0,Y 182.883,Z 577.708,A -85,B 0,C 180,E1 -22592.363,E2 -22592.363} C_VEL
LIN {X 0,Y 179.981,Z 583.435,A -85,B 0,C 180,E1 -22596.727,E2 -22596.727} C_VEL
LIN {X 0,Y 177.879,Z 588.223,A -85,B 0,C 180,E1 -22601.393,E2 -22601.393} C_VEL
LIN {X 0,Y 176.275,Z 592.25,A -85,B 0,C 180,E1 -22606.89,E2 -22606.89} C_VEL
LIN {X 0,Y 175.514,Z 594.975,A -85,B 0,C 180,E1 -22612.932,E2 -22612.932} C_VEL
LIN {X 0,Y 175.524,Z 595.956,A -85,B 0,C 180,E1 -22618.252,E2 -22618.252} C_VEL
LIN {X 0,Y 176.003,Z 595.811,A -85,B 0,C 180,E1 -22623.013,E2 -22623.013} C_VEL
LIN {X 0,Y 177.018,Z 594.724,A -85,B 0,C 180,E1 -22627.435,E2 -22627.435} C_VEL
LIN {X 0,Y 178.756,Z 592.746,A -85,B 0,C 180,E1 -22631.94,E2 -22631.94} C_VEL
LIN {X 0,Y 181.81,Z 589.048,A -85,B 0,C 180,E1 -22637.26,E2 -22637.26} C_VEL
LIN {X 0,Y 186.117,Z 583.815,A -85,B 0,C 180,E1 -22642.463,E2 -22642.463} C_VEL
LIN {X 0,Y 190.49,Z 578.555,A -85,B 0,C 180,E1 -22646.398,E2 -22646.398} C_VEL
LIN {X 0,Y 196.046,Z 571.795,A -85,B 0,C 180,E1 -22650.378,E2 -22650.378} C_VEL
LIN {X 0,Y 202.765,Z 563.135,A -85,B 0,C 180,E1 -22654.311,E2 -22654.311} C_VEL
LIN {X 0,Y 209.235,Z 554.355,A -85,B 0,C 180,E1 -22657.469,E2 -22657.469} C_VEL
LIN {X 0,Y 216.271,Z 544.088,A -85,B 0,C 180,E1 -22660.454,E2 -22660.454} C_VEL
LIN {X 0,Y 223.756,Z 532.211,A -85,B 0,C 180,E1 -22663.178,E2 -22663.178} C_VEL
LIN {X 0,Y 231.261,Z 518.796,A -85,B 0,C 180,E1 -22665.617,E2 -22665.617} C_VEL
LIN {X 0,Y 237.578,Z 506.06,A -85,B 0,C 180,E1 -22667.469,E2 -22667.469} C_VEL
LIN {X 0,Y 243.4,Z 492.836,A -85,B 0,C 180,E1 -22669.023,E2 -22669.023} C_VEL
LIN {X 0,Y 248.767,Z 478.713,A -85,B 0,C 180,E1 -22670.363,E2 -22670.363} C_VEL
LIN {X 0,Y 253.569,Z 463.243,A -85,B 0,C 180,E1 -22671.534,E2 -22671.534} C_VEL
LIN {X 0,Y 257.546,Z 447.502,A -85,B 0,C 180,E1 -22672.419,E2 -22672.419} C_VEL
LIN {X 0,Y 260.714,Z 430.985,A -85,B 0,C 180,E1 -22673.093,E2 -22673.093} C_VEL
LIN {X 0,Y 262.943,Z 413.227,A -85,B 0,C 180,E1 -22673.609,E2 -22673.609} C_VEL
LIN {X 0,Y 270.039,Z 340.526,A -85,B 0,C 180,E1 -22675.392,E2 -22675.392} C_VEL
LIN {X 0,Y 267.074,Z 334.269,A -85,B 0,C 180,E1 -22677.583,E2 -22677.583} C_VEL
LIN {X 0,Y 264.01,Z 328.171,A -85,B 0,C 180,E1 -22680.263,E2 -22680.263} C_VEL
LIN {X 0,Y 261.023,Z 322.439,A -85,B 0,C 180,E1 -22683.663,E2 -22683.663} C_VEL
LIN {X 0,Y 259.802,Z 320.009,A -85,B 0,C 180,E1 -22685.543,E2 -22685.543} C_VEL
LIN {X 0,Y 258.067,Z 317.515,A -85,B 0,C 180,E1 -22689.404,E2 -22689.404} C_VEL
LIN {X 0,Y 257.816,Z 315.525,A -85,B 0,C 180,E1 -22691.92,E2 -22691.92} C_VEL
LIN {X 0,Y 257.763,Z 315.959,A -85,B 0,C 180,E1 -22693.741,E2 -22693.741} C_VEL
LIN {X 0,Y 259.109,Z 319.6,A -85,B 0,C 180,E1 -22698.995,E2 -22698.995} C_VEL
LIN {X 0,Y 259.705,Z 320.472,A -85,B 0,C 180,E1 -22700.036,E2 -22700.036} C_VEL
LIN {X 0,Y 261.773,Z 324.291,A -85,B 0,C 180,E1 -22702.984,E2 -22702.984} C_VEL
LIN {X 0,Y 264.101,Z 328.777,A -85,B 0,C 180,E1 -22705.504,E2 -22705.504} C_VEL
LIN {X 0,Y 267.229,Z 336.178,A -85,B 0,C 180,E1 -22708.309,E2 -22708.309} C_VEL
LIN {X 0,Y 269.879,Z 343.343,A -85,B 0,C 180,E1 -22710.364,E2 -22710.364} C_VEL
LIN {X 0,Y 269.552,Z 346.705,A -85,B 0,C 180,E1 -22710.448,E2 -22710.448} C_VEL
LIN {X 0,Y 268.685,Z 352.556,A -85,B 0,C 180,E1 -22710.437,E2 -22710.437} C_VEL
LIN {X 0,Y 264.653,Z 371.703,A -85,B 0,C 180,E1 -22709.76,E2 -22709.76} C_VEL
LIN {X 0,Y 263.825,Z 377.546,A -85,B 0,C 180,E1 -22709.769,E2 -22709.769} C_VEL
LIN {X 0,Y 258.231,Z 431.22,A -85,B 0,C 180,E1 -22711.093,E2 -22711.093} C_VEL
LIN {X 0,Y 255.114,Z 448.597,A -85,B 0,C 180,E1 -22711.69,E2 -22711.69} C_VEL
LIN {X 0,Y 250.726,Z 465.832,A -85,B 0,C 180,E1 -22712.495,E2 -22712.495} C_VEL
LIN {X 0,Y 246.208,Z 479.968,A -85,B 0,C 180,E1 -22713.392,E2 -22713.392} C_VEL
LIN {X 0,Y 240.328,Z 495.494,A -85,B 0,C 180,E1 -22714.669,E2 -22714.669} C_VEL
LIN {X 0,Y 234.005,Z 509.84,A -85,B 0,C 180,E1 -22716.183,E2 -22716.183} C_VEL
LIN {X 0,Y 226.642,Z 524.242,A -85,B 0,C 180,E1 -22718.109,E2 -22718.109} C_VEL
LIN {X 0,Y 219.036,Z 537.355,A -85,B 0,C 180,E1 -22720.357,E2 -22720.357} C_VEL
LIN {X 0,Y 211.283,Z 549.395,A -85,B 0,C 180,E1 -22722.965,E2 -22722.965} C_VEL
LIN {X 0,Y 203.027,Z 561.122,A -85,B 0,C 180,E1 -22726.187,E2 -22726.187} C_VEL
LIN {X 0,Y 195.636,Z 571.022,A -85,B 0,C 180,E1 -22729.714,E2 -22729.714} C_VEL
LIN {X 0,Y 188.939,Z 579.41,A -85,B 0,C 180,E1 -22733.478,E2 -22733.478} C_VEL
LIN {X 0,Y 181.757,Z 588.136,A -85,B 0,C 180,E1 -22738.659,E2 -22738.659} C_VEL
LIN {X 0,Y 176.384,Z 594.727,A -85,B 0,C 180,E1 -22744.006,E2 -22744.006} C_VEL
LIN {X 0,Y 172.508,Z 599.644,A -85,B 0,C 180,E1 -22749.557,E2 -22749.557} C_VEL
LIN {X 0,Y 170.745,Z 602.089,A -85,B 0,C 180,E1 -22753.255,E2 -22753.255} C_VEL
LIN {X 0,Y 169.358,Z 604.241,A -85,B 0,C 180,E1 -22758.026,E2 -22758.026} C_VEL
LIN {X 0,Y 168.838,Z 605.529,A -85,B 0,C 180,E1 -22762.827,E2 -22762.827} C_VEL
LIN {X 0,Y 168.886,Z 605.771,A -85,B 0,C 180,E1 -22767.616,E2 -22767.616} C_VEL
LIN {X 0,Y 168.998,Z 605.567,A -85,B 0,C 180,E1 -22770.001,E2 -22770.001} C_VEL
LIN {X 0,Y 168.864,Z 604.337,A -85,B 0,C 180,E1 -22774.775,E2 -22774.775} C_VEL
LIN {X 0,Y 169.017,Z 602.093,A -85,B 0,C 180,E1 -22779.575,E2 -22779.575} C_VEL
LIN {X 0,Y 169.908,Z 598.784,A -85,B 0,C 180,E1 -22784.37,E2 -22784.37} C_VEL
LIN {X 0,Y 171.657,Z 594.337,A -85,B 0,C 180,E1 -22789.12,E2 -22789.12} C_VEL
LIN {X 0,Y 174.227,Z 588.753,A -85,B 0,C 180,E1 -22793.79,E2 -22793.79} C_VEL
LIN {X 0,Y 177.809,Z 581.789,A -85,B 0,C 180,E1 -22798.315,E2 -22798.315} C_VEL
LIN {X 0,Y 182.333,Z 573.4,A -85,B 0,C 180,E1 -22802.659,E2 -22802.659} C_VEL
LIN {X 0,Y 187.911,Z 563.381,A -85,B 0,C 180,E1 -22806.756,E2 -22806.756} C_VEL
LIN {X 0,Y 193.481,Z 552.67,A -85,B 0,C 180,E1 -22810.288,E2 -22810.288} C_VEL
LIN {X 0,Y 199.519,Z 540.81,A -85,B 0,C 180,E1 -22813.384,E2 -22813.384} C_VEL
LIN {X 0,Y 204.807,Z 529.552,A -85,B 0,C 180,E1 -22815.752,E2 -22815.752} C_VEL
LIN {X 0,Y 210.897,Z 515.249,A -85,B 0,C 180,E1 -22818.204,E2 -22818.204} C_VEL
LIN {X 0,Y 216.348,Z 501.004,A -85,B 0,C 180,E1 -22820.125,E2 -22820.125} C_VEL
LIN {X 0,Y 221.421,Z 485.598,A -85,B 0,C 180,E1 -22821.774,E2 -22821.774} C_VEL
LIN {X 0,Y 225.761,Z 469.647,A -85,B 0,C 180,E1 -22823.097,E2 -22823.097} C_VEL
LIN {X 0,Y 229.199,Z 453.979,A -85,B 0,C 180,E1 -22824.067,E2 -22824.067} C_VEL
LIN {X 0,Y 232.005,Z 437.582,A -85,B 0,C 180,E1 -22824.78,E2 -22824.78} C_VEL
LIN {X 0,Y 233.943,Z 418.399,A -85,B 0,C 180,E1 -22825.389,E2 -22825.389} C_VEL
LIN {X 0,Y 240.658,Z 334.304,A -85,B 0,C 180,E1 -22827.649,E2 -22827.649} C_VEL
LIN {X 0,Y 233.396,Z 318.615,A -85,B 0,C 180,E1 -22830.781,E2 -22830.781} C_VEL
LIN {X 0,Y 228.713,Z 309.439,A -85,B 0,C 180,E1 -22832.971,E2 -22832.971} C_VEL
LIN {X 0,Y 225.703,Z 304.035,A -85,B 0,C 180,E1 -22834.439,E2 -22834.439} C_VEL
LIN {X 0,Y 218.606,Z 293.136,A -85,B 0,C 180,E1 -22838.169,E2 -22838.169} C_VEL
LIN {X 0,Y 213.012,Z 285.119,A -85,B 0,C 180,E1 -22841.525,E2 -22841.525} C_VEL
LIN {X 0,Y 208.754,Z 279.515,A -85,B 0,C 180,E1 -22844.376,E2 -22844.376} C_VEL
LIN {X 0,Y 205.863,Z 275.551,A -85,B 0,C 180,E1 -22846.585,E2 -22846.585} C_VEL
LIN {X 0,Y 202.944,Z 271.65,A -85,B 0,C 180,E1 -22849.051,E2 -22849.051} C_VEL
LIN {X 0,Y 202.148,Z 270.721,A -85,B 0,C 180,E1 -22849.762,E2 -22849.762} C_VEL
LIN {X 0,Y 199.561,Z 267.584,A -85,B 0,C 180,E1 -22852.284,E2 -22852.284} C_VEL
LIN {X 0,Y 198.493,Z 265.777,A -85,B 0,C 180,E1 -22853.52,E2 -22853.52} C_VEL
LIN {X 0,Y 195.926,Z 263.391,A -85,B 0,C 180,E1 -22856.558,E2 -22856.558} C_VEL
LIN {X 0,Y 194.276,Z 260.241,A -85,B 0,C 180,E1 -22859.159,E2 -22859.159} C_VEL
LIN {X 0,Y 190.856,Z 257.476,A -85,B 0,C 180,E1 -22866.342,E2 -22866.342} C_VEL
LIN {X 0,Y 190.144,Z 255.306,A -85,B 0,C 180,E1 -22870.65,E2 -22870.65} C_VEL
LIN {X 0,Y 189.995,Z 255.303,A -85,B 0,C 180,E1 -22873.912,E2 -22873.912} C_VEL
LIN {X 0,Y 190.297,Z 256.775,A -85,B 0,C 180,E1 -22877.867,E2 -22877.867} C_VEL
LIN {X 0,Y 193.023,Z 260.077,A -85,B 0,C 180,E1 -22885.436,E2 -22885.436} C_VEL
LIN {X 0,Y 194.309,Z 260.815,A -85,B 0,C 180,E1 -22887.495,E2 -22887.495} C_VEL
LIN {X 0,Y 195.987,Z 263.899,A -85,B 0,C 180,E1 -22890.134,E2 -22890.134} C_VEL
LIN {X 0,Y 198.655,Z 266.385,A -85,B 0,C 180,E1 -22893.25,E2 -22893.25} C_VEL
LIN {X 0,Y 200.939,Z 269.832,A -85,B 0,C 180,E1 -22895.698,E2 -22895.698} C_VEL
LIN {X 0,Y 202.754,Z 271.664,A -85,B 0,C 180,E1 -22897.344,E2 -22897.344} C_VEL
LIN {X 0,Y 205.705,Z 275.588,A -85,B 0,C 180,E1 -22899.827,E2 -22899.827} C_VEL
LIN {X 0,Y 207.325,Z 277.807,A -85,B 0,C 180,E1 -22901.107,E2 -22901.107} C_VEL
LIN {X 0,Y 210.635,Z 282.17,A -85,B 0,C 180,E1 -22903.467,E2 -22903.467} C_VEL
LIN {X 0,Y 214.21,Z 287.018,A -85,B 0,C 180,E1 -22905.78,E2 -22905.78} C_VEL
LIN {X 0,Y 219.217,Z 294.164,A -85,B 0,C 180,E1 -22908.703,E2 -22908.703} C_VEL
LIN {X 0,Y 225.43,Z 303.586,A -85,B 0,C 180,E1 -22911.95,E2 -22911.95} C_VEL
LIN {X 0,Y 231.581,Z 313.656,A -85,B 0,C 180,E1 -22914.833,E2 -22914.833} C_VEL
LIN {X 0,Y 239.339,Z 327.355,A -85,B 0,C 180,E1 -22918.107,E2 -22918.107} C_VEL
LIN {X 0,Y 240.753,Z 330.314,A -85,B 0,C 180,E1 -22918.689,E2 -22918.689} C_VEL
LIN {X 0,Y 233.077,Z 423.553,A -85,B 0,C 180,E1 -22921.216,E2 -22921.216} C_VEL
LIN {X 0,Y 230.508,Z 441.185,A -85,B 0,C 180,E1 -22921.969,E2 -22921.969} C_VEL
LIN {X 0,Y 227.169,Z 457.629,A -85,B 0,C 180,E1 -22922.974,E2 -22922.974} C_VEL
LIN {X 0,Y 223.535,Z 472.023,A -85,B 0,C 180,E1 -22924.136,E2 -22924.136} C_VEL
LIN {X 0,Y 219.207,Z 486.576,A -85,B 0,C 180,E1 -22925.62,E2 -22925.62} C_VEL
LIN {X 0,Y 214.11,Z 501.061,A -85,B 0,C 180,E1 -22927.455,E2 -22927.455} C_VEL
LIN {X 0,Y 208.359,Z 515.452,A -85,B 0,C 180,E1 -22929.773,E2 -22929.773} C_VEL
LIN {X 0,Y 202.537,Z 528.257,A -85,B 0,C 180,E1 -22932.324,E2 -22932.324} C_VEL
LIN {X 0,Y 196.359,Z 540.909,A -85,B 0,C 180,E1 -22935.49,E2 -22935.49} C_VEL
LIN {X 0,Y 190.632,Z 551.703,A -85,B 0,C 180,E1 -22938.839,E2 -22938.839} C_VEL
LIN {X 0,Y 185.571,Z 560.942,A -85,B 0,C 180,E1 -22942.382,E2 -22942.382} C_VEL
LIN {X 0,Y 180.587,Z 569.798,A -85,B 0,C 180,E1 -22946.653,E2 -22946.653} C_VEL
LIN {X 0,Y 176.613,Z 577.033,A -85,B 0,C 180,E1 -22951.052,E2 -22951.052} C_VEL
LIN {X 0,Y 173.315,Z 583.248,A -85,B 0,C 180,E1 -22955.818,E2 -22955.818} C_VEL
LIN {X 0,Y 171.276,Z 587.494,A -85,B 0,C 180,E1 -22960.005,E2 -22960.005} C_VEL
LIN {X 0,Y 169.743,Z 590.988,A -85,B 0,C 180,E1 -22964.383,E2 -22964.383} C_VEL
LIN {X 0,Y 168.705,Z 593.831,A -85,B 0,C 180,E1 -22969.466,E2 -22969.466} C_VEL
LIN {X 0,Y 168.334,Z 595.588,A -85,B 0,C 180,E1 -22974.676,E2 -22974.676} C_VEL
LIN {X 0,Y 168.508,Z 596.262,A -85,B 0,C 180,E1 -22980.031,E2 -22980.031} C_VEL
LIN {X 0,Y 169.025,Z 595.989,A -85,B 0,C 180,E1 -22983.737,E2 -22983.737} C_VEL
LIN {X 0,Y 170.182,Z 594.888,A -85,B 0,C 180,E1 -22988.313,E2 -22988.313} C_VEL
LIN {X 0,Y 172.525,Z 592.372,A -85,B 0,C 180,E1 -22993.828,E2 -22993.828} C_VEL
LIN {X 0,Y 176.074,Z 588.44,A -85,B 0,C 180,E1 -22999.32,E2 -22999.32} C_VEL
LIN {X 0,Y 180.974,Z 582.973,A -85,B 0,C 180,E1 -23004.637,E2 -23004.637} C_VEL
LIN {X 0,Y 185.905,Z 577.399,A -85,B 0,C 180,E1 -23008.651,E2 -23008.651} C_VEL
LIN {X 0,Y 192.91,Z 569.223,A -85,B 0,C 180,E1 -23013.195,E2 -23013.195} C_VEL
LIN {X 0,Y 200.042,Z 560.392,A -85,B 0,C 180,E1 -23016.96,E2 -23016.96} C_VEL
LIN {X 0,Y 207.245,Z 550.833,A -85,B 0,C 180,E1 -23020.177,E2 -23020.177} C_VEL
LIN {X 0,Y 214.758,Z 539.979,A -85,B 0,C 180,E1 -23023.049,E2 -23023.049} C_VEL
LIN {X 0,Y 222.383,Z 527.857,A -85,B 0,C 180,E1 -23025.592,E2 -23025.592} C_VEL
LIN {X 0,Y 228.99,Z 516.105,A -85,B 0,C 180,E1 -23027.594,E2 -23027.594} C_VEL
LIN {X 0,Y 235.883,Z 502.303,A -85,B 0,C 180,E1 -23029.481,E2 -23029.481} C_VEL
LIN {X 0,Y 242.437,Z 487.063,A -85,B 0,C 180,E1 -23031.113,E2 -23031.113} C_VEL
LIN {X 0,Y 248.125,Z 471.187,A -85,B 0,C 180,E1 -23032.45,E2 -23032.45} C_VEL
LIN {X 0,Y 252.533,Z 456.062,A -85,B 0,C 180,E1 -23033.431,E2 -23033.431} C_VEL
LIN {X 0,Y 256.083,Z 440.814,A -85,B 0,C 180,E1 -23034.172,E2 -23034.172} C_VEL
LIN {X 0,Y 258.819,Z 424.979,A -85,B 0,C 180,E1 -23034.728,E2 -23034.728} C_VEL
LIN {X 0,Y 267.032,Z 344.837,A -85,B 0,C 180,E1 -23036.698,E2 -23036.698} C_VEL
LIN {X 0,Y 266.637,Z 343.555,A -85,B 0,C 180,E1 -23037.039,E2 -23037.039} C_VEL
LIN {X 0,Y 263.314,Z 336.446,A -85,B 0,C 180,E1 -23039.906,E2 -23039.906} C_VEL
LIN {X 0,Y 261.538,Z 332.939,A -85,B 0,C 180,E1 -23041.76,E2 -23041.76} C_VEL
LIN {X 0,Y 259.502,Z 328.739,A -85,B 0,C 180,E1 -23044.411,E2 -23044.411} C_VEL
LIN {X 0,Y 258.595,Z 326.885,A -85,B 0,C 180,E1 -23045.905,E2 -23045.905} C_VEL
LIN {X 0,Y 257.007,Z 324.267,A -85,B 0,C 180,E1 -23049.881,E2 -23049.881} C_VEL
LIN {X 0,Y 256.839,Z 322.56,A -85,B 0,C 180,E1 -23052.175,E2 -23052.175} C_VEL
LIN {X 0,Y 256.797,Z 323.014,A -85,B 0,C 180,E1 -23053.638,E2 -23053.638} C_VEL
LIN {X 0,Y 258.181,Z 326.711,A -85,B 0,C 180,E1 -23059.066,E2 -23059.066} C_VEL
LIN {X 0,Y 260.407,Z 331.011,A -85,B 0,C 180,E1 -23062.567,E2 -23062.567} C_VEL
LIN {X 0,Y 262.502,Z 335.226,A -85,B 0,C 180,E1 -23064.95,E2 -23064.95} C_VEL
LIN {X 0,Y 265.271,Z 342.188,A -85,B 0,C 180,E1 -23067.613,E2 -23067.613} C_VEL
LIN {X 0,Y 266.903,Z 346.896,A -85,B 0,C 180,E1 -23069.022,E2 -23069.022} C_VEL
LIN {X 0,Y 263.825,Z 377.546,A -85,B 0,C 180,E1 -23069.769,E2 -23069.769} C_VEL
LIN {X 0,Y 262.985,Z 383.395,A -85,B 0,C 180,E1 -23069.77,E2 -23069.77} C_VEL
LIN {X 0,Y 258.941,Z 402.522,A -85,B 0,C 180,E1 -23069.032,E2 -23069.032} C_VEL
LIN {X 0,Y 258.109,Z 408.366,A -85,B 0,C 180,E1 -23069.039,E2 -23069.039} C_VEL
LIN {X 0,Y 255.22,Z 433.074,A -85,B 0,C 180,E1 -23069.674,E2 -23069.674} C_VEL
LIN {X 0,Y 252.021,Z 449.896,A -85,B 0,C 180,E1 -23070.259,E2 -23070.259} C_VEL
LIN {X 0,Y 247.716,Z 466.252,A -85,B 0,C 180,E1 -23071.019,E2 -23071.019} C_VEL
LIN {X 0,Y 242.477,Z 482.016,A -85,B 0,C 180,E1 -23072.03,E2 -23072.03} C_VEL
LIN {X 0,Y 237.082,Z 495.557,A -85,B 0,C 180,E1 -23073.132,E2 -23073.132} C_VEL
LIN {X 0,Y 230.581,Z 509.795,A -85,B 0,C 180,E1 -23074.621,E2 -23074.621} C_VEL
LIN {X 0,Y 222.969,Z 524.134,A -85,B 0,C 180,E1 -23076.511,E2 -23076.511} C_VEL
LIN {X 0,Y 214.543,Z 538.185,A -85,B 0,C 180,E1 -23078.924,E2 -23078.924} C_VEL
LIN {X 0,Y 207.628,Z 548.458,A -85,B 0,C 180,E1 -23081.138,E2 -23081.138} C_VEL
LIN {X 0,Y 200.05,Z 558.922,A -85,B 0,C 180,E1 -23083.932,E2 -23083.932} C_VEL
LIN {X 0,Y 191.98,Z 569.266,A -85,B 0,C 180,E1 -23087.463,E2 -23087.463} C_VEL
LIN {X 0,Y 184.902,Z 577.692,A -85,B 0,C 180,E1 -23091.161,E2 -23091.161} C_VEL
LIN {X 0,Y 178.612,Z 584.939,A -85,B 0,C 180,E1 -23095.213,E2 -23095.213} C_VEL
LIN {X 0,Y 173.273,Z 590.976,A -85,B 0,C 180,E1 -23099.537,E2 -23099.537} C_VEL
LIN {X 0,Y 168.954,Z 595.86,A -85,B 0,C 180,E1 -23104.103,E2 -23104.103} C_VEL
LIN {X 0,Y 165.033,Z 600.544,A -85,B 0,C 180,E1 -23110.083,E2 -23110.083} C_VEL
LIN {X 0,Y 162.979,Z 603.183,A -85,B 0,C 180,E1 -23115.006,E2 -23115.006} C_VEL
LIN {X 0,Y 161.951,Z 604.839,A -85,B 0,C 180,E1 -23120.005,E2 -23120.005} C_VEL
LIN {X 0,Y 161.732,Z 605.566,A -85,B 0,C 180,E1 -23125.015,E2 -23125.015} C_VEL
LIN {X 0,Y 161.909,Z 605.311,A -85,B 0,C 180,E1 -23130.001,E2 -23130.001} C_VEL
LIN {X 0,Y 161.812,Z 604.802,A -85,B 0,C 180,E1 -23132.616,E2 -23132.616} C_VEL
LIN {X 0,Y 161.807,Z 603.011,A -85,B 0,C 180,E1 -23137.488,E2 -23137.488} C_VEL
LIN {X 0,Y 162.336,Z 600.214,A -85,B 0,C 180,E1 -23142.502,E2 -23142.502} C_VEL
LIN {X 0,Y 163.803,Z 596.263,A -85,B 0,C 180,E1 -23147.478,E2 -23147.478} C_VEL
LIN {X 0,Y 166.102,Z 591.182,A -85,B 0,C 180,E1 -23152.384,E2 -23152.384} C_VEL
LIN {X 0,Y 169.414,Z 584.889,A -85,B 0,C 180,E1 -23157.151,E2 -23157.151} C_VEL
LIN {X 0,Y 173.995,Z 576.676,A -85,B 0,C 180,E1 -23161.981,E2 -23161.981} C_VEL
LIN {X 0,Y 179.077,Z 567.872,A -85,B 0,C 180,E1 -23166.064,E2 -23166.064} C_VEL
LIN {X 0,Y 184.515,Z 558.317,A -85,B 0,C 180,E1 -23169.642,E2 -23169.642} C_VEL
LIN {X 0,Y 190.556,Z 547.106,A -85,B 0,C 180,E1 -23173.024,E2 -23173.024} C_VEL
LIN {X 0,Y 197.226,Z 533.805,A -85,B 0,C 180,E1 -23176.186,E2 -23176.186} C_VEL
LIN {X 0,Y 203.497,Z 520.286,A -85,B 0,C 180,E1 -23178.691,E2 -23178.691} C_VEL
LIN {X 0,Y 208.962,Z 506.987,A -85,B 0,C 180,E1 -23180.674,E2 -23180.674} C_VEL
LIN {X 0,Y 214.085,Z 492.857,A -85,B 0,C 180,E1 -23182.371,E2 -23182.371} C_VEL
LIN {X 0,Y 218.797,Z 477.672,A -85,B 0,C 180,E1 -23183.808,E2 -23183.808} C_VEL
LIN {X 0,Y 222.676,Z 462.123,A -85,B 0,C 180,E1 -23184.947,E2 -23184.947} C_VEL
LIN {X 0,Y 225.985,Z 445.989,A -85,B 0,C 180,E1 -23185.786,E2 -23185.786} C_VEL
LIN {X 0,Y 228.302,Z 430.157,A -85,B 0,C 180,E1 -23186.379,E2 -23186.379} C_VEL
LIN {X 0,Y 236.074,Z 337.094,A -85,B 0,C 180,E1 -23188.914,E2 -23188.914} C_VEL
LIN {X 0,Y 229.287,Z 322.224,A -85,B 0,C 180,E1 -23192.008,E2 -23192.008} C_VEL
LIN {X 0,Y 223.407,Z 310.666,A -85,B 0,C 180,E1 -23194.932,E2 -23194.932} C_VEL
LIN {X 0,Y 217.502,Z 301.43,A -85,B 0,C 180,E1 -23198.092,E2 -23198.092} C_VEL
LIN {X 0,Y 212.251,Z 293.537,A -85,B 0,C 180,E1 -23201.258,E2 -23201.258} C_VEL
LIN {X 0,Y 209.34,Z 289.568,A -85,B 0,C 180,E1 -23203.168,E2 -23203.168} C_VEL
LIN {X 0,Y 206.941,Z 286.11,A -85,B 0,C 180,E1 -23204.893,E2 -23204.893} C_VEL
LIN {X 0,Y 203.825,Z 281.824,A -85,B 0,C 180,E1 -23207.37,E2 -23207.37} C_VEL
LIN {X 0,Y 200.727,Z 277.566,A -85,B 0,C 180,E1 -23210.113,E2 -23210.113} C_VEL
LIN {X 0,Y 198.084,Z 274.369,A -85,B 0,C 180,E1 -23212.765,E2 -23212.765} C_VEL
LIN {X 0,Y 196.98,Z 272.537,A -85,B 0,C 180,E1 -23214.067,E2 -23214.067} C_VEL
LIN {X 0,Y 194.325,Z 269.808,A -85,B 0,C 180,E1 -23217.392,E2 -23217.392} C_VEL
LIN {X 0,Y 193.036,Z 267.151,A -85,B 0,C 180,E1 -23219.577,E2 -23219.577} C_VEL
LIN {X 0,Y 189.793,Z 264.36,A -85,B 0,C 180,E1 -23226.752,E2 -23226.752} C_VEL
LIN {X 0,Y 189.182,Z 262.387,A -85,B 0,C 180,E1 -23230.705,E2 -23230.705} C_VEL
LIN {X 0,Y 189.042,Z 262.269,A -85,B 0,C 180,E1 -23233.436,E2 -23233.436} C_VEL
LIN {X 0,Y 189.29,Z 263.705,A -85,B 0,C 180,E1 -23237.515,E2 -23237.515} C_VEL
LIN {X 0,Y 192.135,Z 267.164,A -85,B 0,C 180,E1 -23245.562,E2 -23245.562} C_VEL
LIN {X 0,Y 193.065,Z 267.782,A -85,B 0,C 180,E1 -23247.099,E2 -23247.099} C_VEL
LIN {X 0,Y 194.965,Z 271.087,A -85,B 0,C 180,E1 -23250.101,E2 -23250.101} C_VEL
LIN {X 0,Y 197.148,Z 273.135,A -85,B 0,C 180,E1 -23252.717,E2 -23252.717} C_VEL
LIN {X 0,Y 199.522,Z 276.659,A -85,B 0,C 180,E1 -23255.316,E2 -23255.316} C_VEL
LIN {X 0,Y 201.224,Z 278.555,A -85,B 0,C 180,E1 -23256.925,E2 -23256.925} C_VEL
LIN {X 0,Y 204.131,Z 282.379,A -85,B 0,C 180,E1 -23259.43,E2 -23259.43} C_VEL
LIN {X 0,Y 208.473,Z 288.429,A -85,B 0,C 180,E1 -23262.758,E2 -23262.758} C_VEL
LIN {X 0,Y 211.809,Z 293.028,A -85,B 0,C 180,E1 -23264.989,E2 -23264.989} C_VEL
LIN {X 0,Y 216.598,Z 300.06,A -85,B 0,C 180,E1 -23267.921,E2 -23267.921} C_VEL
LIN {X 0,Y 223.429,Z 310.659,A -85,B 0,C 180,E1 -23271.599,E2 -23271.599} C_VEL
LIN {X 0,Y 229.629,Z 321.231,A -85,B 0,C 180,E1 -23274.575,E2 -23274.575} C_VEL
LIN {X 0,Y 236.114,Z 333.114,A -85,B 0,C 180,E1 -23277.407,E2 -23277.407} C_VEL
LIN {X 0,Y 228.582,Z 422.742,A -85,B 0,C 180,E1 -23279.85,E2 -23279.85} C_VEL
LIN {X 0,Y 226.101,Z 439.698,A -85,B 0,C 180,E1 -23280.554,E2 -23280.554} C_VEL
LIN {X 0,Y 222.9,Z 455.661,A -85,B 0,C 180,E1 -23281.498,E2 -23281.498} C_VEL
LIN {X 0,Y 218.81,Z 471.717,A -85,B 0,C 180,E1 -23282.761,E2 -23282.761} C_VEL
LIN {X 0,Y 214.341,Z 486.385,A -85,B 0,C 180,E1 -23284.249,E2 -23284.249} C_VEL
LIN {X 0,Y 208.834,Z 501.549,A -85,B 0,C 180,E1 -23286.181,E2 -23286.181} C_VEL
LIN {X 0,Y 203.114,Z 515.37,A -85,B 0,C 180,E1 -23288.43,E2 -23288.43} C_VEL
LIN {X 0,Y 197.582,Z 527.221,A -85,B 0,C 180,E1 -23290.79,E2 -23290.79} C_VEL
LIN {X 0,Y 191.983,Z 538.422,A -85,B 0,C 180,E1 -23293.518,E2 -23293.518} C_VEL
LIN {X 0,Y 185.948,Z 549.588,A -85,B 0,C 180,E1 -23296.892,E2 -23296.892} C_VEL
LIN {X 0,Y 179.782,Z 560.357,A -85,B 0,C 180,E1 -23301.003,E2 -23301.003} C_VEL
LIN {X 0,Y 174.487,Z 569.357,A -85,B 0,C 180,E1 -23305.379,E2 -23305.379} C_VEL
LIN {X 0,Y 170.128,Z 576.854,A -85,B 0,C 180,E1 -23309.999,E2 -23309.999} C_VEL
LIN {X 0,Y 166.7,Z 583.05,A -85,B 0,C 180,E1 -23314.836,E2 -23314.836} C_VEL
LIN {X 0,Y 164.131,Z 588.07,A -85,B 0,C 180,E1 -23319.987,E2 -23319.987} C_VEL
LIN {X 0,Y 162.436,Z 591.74,A -85,B 0,C 180,E1 -23325.045,E2 -23325.045} C_VEL
LIN {X 0,Y 161.486,Z 594.462,A -85,B 0,C 180,E1 -23330.374,E2 -23330.374} C_VEL
LIN {X 0,Y 161.285,Z 595.574,A -85,B 0,C 180,E1 -23333.784,E2 -23333.784} C_VEL
LIN {X 0,Y 161.369,Z 596.414,A -85,B 0,C 180,E1 -23339.42,E2 -23339.42} C_VEL
LIN {X 0,Y 162.062,Z 596.17,A -85,B 0,C 180,E1 -23344.518,E2 -23344.518} C_VEL
LIN {X 0,Y 163.667,Z 594.808,A -85,B 0,C 180,E1 -23350.097,E2 -23350.097} C_VEL
LIN {X 0,Y 166.467,Z 592.015,A -85,B 0,C 180,E1 -23355.864,E2 -23355.864} C_VEL
LIN {X 0,Y 170.58,Z 587.796,A -85,B 0,C 180,E1 -23361.517,E2 -23361.517} C_VEL
LIN {X 0,Y 176.098,Z 582.04,A -85,B 0,C 180,E1 -23366.938,E2 -23366.938} C_VEL
LIN {X 0,Y 182.142,Z 575.671,A -85,B 0,C 180,E1 -23371.377,E2 -23371.377} C_VEL
LIN {X 0,Y 188.518,Z 568.543,A -85,B 0,C 180,E1 -23375.197,E2 -23375.197} C_VEL
LIN {X 0,Y 196.307,Z 559.312,A -85,B 0,C 180,E1 -23379.022,E2 -23379.022} C_VEL
LIN {X 0,Y 204.139,Z 549.246,A -85,B 0,C 180,E1 -23382.296,E2 -23382.296} C_VEL
LIN {X 0,Y 211.862,Z 538.481,A -85,B 0,C 180,E1 -23385.045,E2 -23385.045} C_VEL
LIN {X 0,Y 219.778,Z 526.114,A -85,B 0,C 180,E1 -23387.556,E2 -23387.556} C_VEL
LIN {X 0,Y 227.519,Z 512.432,A -85,B 0,C 180,E1 -23389.737,E2 -23389.737} C_VEL
LIN {X 0,Y 234.485,Z 498.328,A -85,B 0,C 180,E1 -23391.516,E2 -23391.516} C_VEL
LIN {X 0,Y 240.753,Z 483.58,A -85,B 0,C 180,E1 -23392.977,E2 -23392.977} C_VEL
LIN {X 0,Y 246.096,Z 468.599,A -85,B 0,C 180,E1 -23394.148,E2 -23394.148} C_VEL
LIN {X 0,Y 250.564,Z 453.07,A -85,B 0,C 180,E1 -23395.105,E2 -23395.105} C_VEL
LIN {X 0,Y 254.355,Z 435.9,A -85,B 0,C 180,E1 -23395.849,E2 -23395.849} C_VEL
LIN {X 0,Y 256.851,Z 419.403,A -85,B 0,C 180,E1 -23396.348,E2 -23396.348} C_VEL
LIN {X 0,Y 264.28,Z 348.648,A -85,B 0,C 180,E1 -23398.059,E2 -23398.059} C_VEL
LIN {X 0,Y 261.133,Z 341.643,A -85,B 0,C 180,E1 -23401.066,E2 -23401.066} C_VEL
LIN {X 0,Y 258.327,Z 335.652,A -85,B 0,C 180,E1 -23404.682,E2 -23404.682} C_VEL
LIN {X 0,Y 257.398,Z 333.756,A -85,B 0,C 180,E1 -23406.27,E2 -23406.27} C_VEL
LIN {X 0,Y 255.981,Z 331.051,A -85,B 0,C 180,E1 -23410.305,E2 -23410.305} C_VEL
LIN {X 0,Y 255.889,Z 329.703,A -85,B 0,C 180,E1 -23411.985,E2 -23411.985} C_VEL
LIN {X 0,Y 255.841,Z 329.808,A -85,B 0,C 180,E1 -23413.198,E2 -23413.198} C_VEL
LIN {X 0,Y 257.012,Z 333.547,A -85,B 0,C 180,E1 -23418.655,E2 -23418.655} C_VEL
LIN {X 0,Y 257.673,Z 334.946,A -85,B 0,C 180,E1 -23419.969,E2 -23419.969} C_VEL
LIN {X 0,Y 259.086,Z 337.78,A -85,B 0,C 180,E1 -23422.163,E2 -23422.163} C_VEL
LIN {X 0,Y 261.022,Z 341.881,A -85,B 0,C 180,E1 -23424.493,E2 -23424.493} C_VEL
LIN {X 0,Y 263.418,Z 348.414,A -85,B 0,C 180,E1 -23426.972,E2 -23426.972} C_VEL
LIN {X 0,Y 264.145,Z 350.671,A -85,B 0,C 180,E1 -23427.664,E2 -23427.664} C_VEL
LIN {X 0,Y 258.109,Z 408.366,A -85,B 0,C 180,E1 -23429.039,E2 -23429.039} C_VEL
LIN {X 0,Y 257.284,Z 414.221,A -85,B 0,C 180,E1 -23429.043,E2 -23429.043} C_VEL
LIN {X 0,Y 252.957,Z 433.323,A -85,B 0,C 180,E1 -23428.306,E2 -23428.306} C_VEL
LIN {X 0,Y 251.756,Z 439.11,A -85,B 0,C 180,E1 -23428.355,E2 -23428.355} C_VEL
LIN {X 0,Y 247.931,Z 456.027,A -85,B 0,C 180,E1 -23428.997,E2 -23428.997} C_VEL
LIN {X 0,Y 243.405,Z 471.287,A -85,B 0,C 180,E1 -23429.784,E2 -23429.784} C_VEL
LIN {X 0,Y 238.174,Z 485.767,A -85,B 0,C 180,E1 -23430.751,E2 -23430.751} C_VEL
LIN {X 0,Y 232.71,Z 498.683,A -85,B 0,C 180,E1 -23431.857,E2 -23431.857} C_VEL
LIN {X 0,Y 226.026,Z 512.337,A -85,B 0,C 180,E1 -23433.319,E2 -23433.319} C_VEL
LIN {X 0,Y 218.248,Z 526.224,A -85,B 0,C 180,E1 -23435.204,E2 -23435.204} C_VEL
LIN {X 0,Y 210.19,Z 539.004,A -85,B 0,C 180,E1 -23437.43,E2 -23437.43} C_VEL
LIN {X 0,Y 201.915,Z 550.719,A -85,B 0,C 180,E1 -23440.028,E2 -23440.028} C_VEL
LIN {X 0,Y 194.116,Z 560.777,A -85,B 0,C 180,E1 -23442.85,E2 -23442.85} C_VEL
LIN {X 0,Y 185.935,Z 570.63,A -85,B 0,C 180,E1 -23446.386,E2 -23446.386} C_VEL
LIN {X 0,Y 179.396,Z 577.984,A -85,B 0,C 180,E1 -23449.731,E2 -23449.731} C_VEL
LIN {X 0,Y 172.766,Z 585.128,A -85,B 0,C 180,E1 -23453.855,E2 -23453.855} C_VEL
LIN {X 0,Y 167.111,Z 591.118,A -85,B 0,C 180,E1 -23458.286,E2 -23458.286} C_VEL
LIN {X 0,Y 161.532,Z 596.98,A -85,B 0,C 180,E1 -23464.211,E2 -23464.211} C_VEL
LIN {X 0,Y 158.287,Z 600.499,A -85,B 0,C 180,E1 -23469.195,E2 -23469.195} C_VEL
LIN {X 0,Y 156.075,Z 603.102,A -85,B 0,C 180,E1 -23474.326,E2 -23474.326} C_VEL
LIN {X 0,Y 154.909,Z 604.683,A -85,B 0,C 180,E1 -23479.545,E2 -23479.545} C_VEL
LIN {X 0,Y 154.633,Z 605.376,A -85,B 0,C 180,E1 -23484.785,E2 -23484.785} C_VEL
LIN {X 0,Y 154.81,Z 605.056,A -85,B 0,C 180,E1 -23490.001,E2 -23490.001} C_VEL
LIN {X 0,Y 154.735,Z 604.554,A -85,B 0,C 180,E1 -23492.604,E2 -23492.604} C_VEL
LIN {X 0,Y 154.722,Z 602.687,A -85,B 0,C 180,E1 -23497.833,E2 -23497.833} C_VEL
LIN {X 0,Y 155.336,Z 599.819,A -85,B 0,C 180,E1 -23503.075,E2 -23503.075} C_VEL
LIN {X 0,Y 156.958,Z 595.831,A -85,B 0,C 180,E1 -23508.267,E2 -23508.267} C_VEL
LIN {X 0,Y 159.45,Z 590.671,A -85,B 0,C 180,E1 -23513.372,E2 -23513.372} C_VEL
LIN {X 0,Y 163.01,Z 584.316,A -85,B 0,C 180,E1 -23518.311,E2 -23518.311} C_VEL
LIN {X 0,Y 168.268,Z 575.456,A -85,B 0,C 180,E1 -23523.602,E2 -23523.602} C_VEL
LIN {X 0,Y 174.062,Z 565.862,A -85,B 0,C 180,E1 -23528.006,E2 -23528.006} C_VEL
LIN {X 0,Y 179.846,Z 555.92,A -85,B 0,C 180,E1 -23531.631,E2 -23531.631} C_VEL
LIN {X 0,Y 186.283,Z 544.286,A -85,B 0,C 180,E1 -23535.023,E2 -23535.023} C_VEL
LIN {X 0,Y 192.855,Z 531.592,A -85,B 0,C 180,E1 -23537.945,E2 -23537.945} C_VEL
LIN {X 0,Y 198.803,Z 518.995,A -85,B 0,C 180,E1 -23540.255,E2 -23540.255} C_VEL
LIN {X 0,Y 204.426,Z 505.439,A -85,B 0,C 180,E1 -23542.253,E2 -23542.253} C_VEL
LIN {X 0,Y 209.745,Z 490.994,A -85,B 0,C 180,E1 -23543.936,E2 -23543.936} C_VEL
LIN {X 0,Y 214.602,Z 475.388,A -85,B 0,C 180,E1 -23545.368,E2 -23545.368} C_VEL
LIN {X 0,Y 218.646,Z 459.483,A -85,B 0,C 180,E1 -23546.482,E2 -23546.482} C_VEL
LIN {X 0,Y 222.042,Z 442.348,A -85,B 0,C 180,E1 -23547.321,E2 -23547.321} C_VEL
LIN {X 0,Y 223.971,Z 427.757,A -85,B 0,C 180,E1 -23547.842,E2 -23547.842} C_VEL
LIN {X 0,Y 231.55,Z 339.914,A -85,B 0,C 180,E1 -23550.219,E2 -23550.219} C_VEL
LIN {X 0,Y 225.278,Z 325.913,A -85,B 0,C 180,E1 -23553.262,E2 -23553.262} C_VEL
LIN {X 0,Y 220.198,Z 315.76,A -85,B 0,C 180,E1 -23555.925,E2 -23555.925} C_VEL
LIN {X 0,Y 213.204,Z 304.607,A -85,B 0,C 180,E1 -23559.907,E2 -23559.907} C_VEL
LIN {X 0,Y 208.171,Z 297.105,A -85,B 0,C 180,E1 -23563.197,E2 -23563.197} C_VEL
LIN {X 0,Y 204.588,Z 292.044,A -85,B 0,C 180,E1 -23565.843,E2 -23565.843} C_VEL
LIN {X 0,Y 201.925,Z 288.241,A -85,B 0,C 180,E1 -23568.048,E2 -23568.048} C_VEL
LIN {X 0,Y 198.806,Z 283.928,A -85,B 0,C 180,E1 -23570.945,E2 -23570.945} C_VEL
LIN {X 0,Y 196.19,Z 280.402,A -85,B 0,C 180,E1 -23573.758,E2 -23573.758} C_VEL
LIN {X 0,Y 195.491,Z 279.293,A -85,B 0,C 180,E1 -23574.614,E2 -23574.614} C_VEL
LIN {X 0,Y 192.908,Z 276.421,A -85,B 0,C 180,E1 -23578.02,E2 -23578.02} C_VEL
LIN {X 0,Y 191.802,Z 274.052,A -85,B 0,C 180,E1 -23580,E2 -23580} C_VEL
LIN {X 0,Y 188.831,Z 271.405,A -85,B 0,C 180,E1 -23586.786,E2 -23586.786} C_VEL
LIN {X 0,Y 188.224,Z 269.434,A -85,B 0,C 180,E1 -23590.76,E2 -23590.76} C_VEL
LIN {X 0,Y 188.098,Z 269.358,A -85,B 0,C 180,E1 -23593.724,E2 -23593.724} C_VEL
LIN {X 0,Y 188.394,Z 271.027,A -85,B 0,C 180,E1 -23597.935,E2 -23597.935} C_VEL
LIN {X 0,Y 191.247,Z 274.25,A -85,B 0,C 180,E1 -23605.689,E2 -23605.689} C_VEL
LIN {X 0,Y 191.825,Z 274.715,A -85,B 0,C 180,E1 -23606.683,E2 -23606.683} C_VEL
LIN {X 0,Y 193.918,Z 278.224,A -85,B 0,C 180,E1 -23610.031,E2 -23610.031} C_VEL
LIN {X 0,Y 195.742,Z 280.033,A -85,B 0,C 180,E1 -23612.283,E2 -23612.283} C_VEL
LIN {X 0,Y 198.181,Z 283.558,A -85,B 0,C 180,E1 -23614.997,E2 -23614.997} C_VEL
LIN {X 0,Y 199.488,Z 285.11,A -85,B 0,C 180,E1 -23616.285,E2 -23616.285} C_VEL
LIN {X 0,Y 203.188,Z 290.236,A -85,B 0,C 180,E1 -23619.564,E2 -23619.564} C_VEL
LIN {X 0,Y 206.497,Z 294.9,A -85,B 0,C 180,E1 -23622.148,E2 -23622.148} C_VEL
LIN {X 0,Y 209.892,Z 299.739,A -85,B 0,C 180,E1 -23624.5,E2 -23624.5} C_VEL
LIN {X 0,Y 214.052,Z 306.015,A -85,B 0,C 180,E1 -23627.142,E2 -23627.142} C_VEL
LIN {X 0,Y 220.607,Z 316.406,A -85,B 0,C 180,E1 -23630.812,E2 -23630.812} C_VEL
LIN {X 0,Y 226.975,Z 327.591,A -85,B 0,C 180,E1 -23633.984,E2 -23633.984} C_VEL
LIN {X 0,Y 231.62,Z 336.169,A -85,B 0,C 180,E1 -23636.112,E2 -23636.112} C_VEL
LIN {X 0,Y 223.973,Z 423.595,A -85,B 0,C 180,E1 -23638.49,E2 -23638.49} C_VEL
LIN {X 0,Y 221.309,Z 441.102,A -85,B 0,C 180,E1 -23639.235,E2 -23639.235} C_VEL
LIN {X 0,Y 217.906,Z 457.067,A -85,B 0,C 180,E1 -23640.192,E2 -23640.192} C_VEL
LIN {X 0,Y 213.601,Z 473.269,A -85,B 0,C 180,E1 -23641.504,E2 -23641.504} C_VEL
LIN {X 0,Y 208.457,Z 489.253,A -85,B 0,C 180,E1 -23643.196,E2 -23643.196} C_VEL
LIN {X 0,Y 202.803,Z 503.969,A -85,B 0,C 180,E1 -23645.154,E2 -23645.154} C_VEL
LIN {X 0,Y 196.933,Z 517.548,A -85,B 0,C 180,E1 -23647.44,E2 -23647.44} C_VEL
LIN {X 0,Y 190.746,Z 530.122,A -85,B 0,C 180,E1 -23650.073,E2 -23650.073} C_VEL
LIN {X 0,Y 184.3,Z 542.219,A -85,B 0,C 180,E1 -23653.265,E2 -23653.265} C_VEL
LIN {X 0,Y 178.007,Z 553.149,A -85,B 0,C 180,E1 -23656.878,E2 -23656.878} C_VEL
LIN {X 0,Y 171.909,Z 563.244,A -85,B 0,C 180,E1 -23661.103,E2 -23661.103} C_VEL
LIN {X 0,Y 167.183,Z 571.001,A -85,B 0,C 180,E1 -23665.176,E2 -23665.176} C_VEL
LIN {X 0,Y 162.794,Z 578.218,A -85,B 0,C 180,E1 -23669.999,E2 -23669.999} C_VEL
LIN {X 0,Y 159.314,Z 584.162,A -85,B 0,C 180,E1 -23675.061,E2 -23675.061} C_VEL
LIN {X 0,Y 156.826,Z 588.937,A -85,B 0,C 180,E1 -23680.326,E2 -23680.326} C_VEL
LIN {X 0,Y 155.145,Z 592.492,A -85,B 0,C 180,E1 -23685.77,E2 -23685.77} C_VEL
LIN {X 0,Y 154.282,Z 594.984,A -85,B 0,C 180,E1 -23691.371,E2 -23691.371} C_VEL
LIN {X 0,Y 154.167,Z 595.84,A -85,B 0,C 180,E1 -23694.254,E2 -23694.254} C_VEL
LIN {X 0,Y 154.334,Z 596.641,A -85,B 0,C 180,E1 -23700.093,E2 -23700.093} C_VEL
LIN {X 0,Y 155.255,Z 596.245,A -85,B 0,C 180,E1 -23706.047,E2 -23706.047} C_VEL
LIN {X 0,Y 157.306,Z 594.612,A -85,B 0,C 180,E1 -23712.078,E2 -23712.078} C_VEL
LIN {X 0,Y 160.619,Z 591.638,A -85,B 0,C 180,E1 -23718.058,E2 -23718.058} C_VEL
LIN {X 0,Y 165.339,Z 587.172,A -85,B 0,C 180,E1 -23723.863,E2 -23723.863} C_VEL
LIN {X 0,Y 170.082,Z 582.55,A -85,B 0,C 180,E1 -23728.218,E2 -23728.218} C_VEL
LIN {X 0,Y 175.205,Z 577.499,A -85,B 0,C 180,E1 -23731.941,E2 -23731.941} C_VEL
LIN {X 0,Y 182.387,Z 570.013,A -85,B 0,C 180,E1 -23736.225,E2 -23736.225} C_VEL
LIN {X 0,Y 190.518,Z 561.021,A -85,B 0,C 180,E1 -23740.144,E2 -23740.144} C_VEL
LIN {X 0,Y 198.856,Z 550.888,A -85,B 0,C 180,E1 -23743.576,E2 -23743.576} C_VEL
LIN {X 0,Y 207.467,Z 539.441,A -85,B 0,C 180,E1 -23746.548,E2 -23746.548} C_VEL
LIN {X 0,Y 215.643,Z 527.216,A -85,B 0,C 180,E1 -23749.045,E2 -23749.045} C_VEL
LIN {X 0,Y 223.453,Z 514.048,A -85,B 0,C 180,E1 -23751.162,E2 -23751.162} C_VEL
LIN {X 0,Y 230.198,Z 501.092,A -85,B 0,C 180,E1 -23752.826,E2 -23752.826} C_VEL
LIN {X 0,Y 237.022,Z 485.926,A -85,B 0,C 180,E1 -23754.354,E2 -23754.354} C_VEL
LIN {X 0,Y 242.75,Z 470.744,A -85,B 0,C 180,E1 -23755.561,E2 -23755.561} C_VEL
LIN {X 0,Y 247.662,Z 454.433,A -85,B 0,C 180,E1 -23756.566,E2 -23756.566} C_VEL
LIN {X 0,Y 251.476,Z 438.11,A -85,B 0,C 180,E1 -23757.281,E2 -23757.281} C_VEL
LIN {X 0,Y 254.294,Z 420.906,A -85,B 0,C 180,E1 -23757.808,E2 -23757.808} C_VEL
LIN {X 0,Y 261.649,Z 353.097,A -85,B 0,C 180,E1 -23759.417,E2 -23759.417} C_VEL
LIN {X 0,Y 259.359,Z 347.571,A -85,B 0,C 180,E1 -23761.887,E2 -23761.887} C_VEL
LIN {X 0,Y 256.906,Z 341.996,A -85,B 0,C 180,E1 -23765.383,E2 -23765.383} C_VEL
LIN {X 0,Y 256.211,Z 340.583,A -85,B 0,C 180,E1 -23766.695,E2 -23766.695} C_VEL
LIN {X 0,Y 254.947,Z 337.724,A -85,B 0,C 180,E1 -23770.939,E2 -23770.939} C_VEL
LIN {X 0,Y 254.921,Z 336.805,A -85,B 0,C 180,E1 -23772.031,E2 -23772.031} C_VEL
LIN {X 0,Y 254.885,Z 336.788,A -85,B 0,C 180,E1 -23772.996,E2 -23772.996} C_VEL
LIN {X 0,Y 255.847,Z 340.401,A -85,B 0,C 180,E1 -23778.228,E2 -23778.228} C_VEL
LIN {X 0,Y 256.363,Z 341.471,A -85,B 0,C 180,E1 -23779.382,E2 -23779.382} C_VEL
LIN {X 0,Y 257.834,Z 344.635,A -85,B 0,C 180,E1 -23781.82,E2 -23781.82} C_VEL
LIN {X 0,Y 259.423,Z 348.215,A -85,B 0,C 180,E1 -23783.872,E2 -23783.872} C_VEL
LIN {X 0,Y 261.55,Z 354.477,A -85,B 0,C 180,E1 -23786.274,E2 -23786.274} C_VEL
LIN {X 0,Y 253.362,Z 429.528,A -85,B 0,C 180,E1 -23788.078,E2 -23788.078} C_VEL
LIN {X 0,Y 251.756,Z 439.11,A -85,B 0,C 180,E1 -23788.355,E2 -23788.355} C_VEL
LIN {X 0,Y 250.413,Z 444.868,A -85,B 0,C 180,E1 -23788.406,E2 -23788.406} C_VEL
LIN {X 0,Y 247.243,Z 454.211,A -85,B 0,C 180,E1 -23788.129,E2 -23788.129} C_VEL
LIN {X 0,Y 243.677,Z 463.4,A -85,B 0,C 180,E1 -23787.912,E2 -23787.912} C_VEL
LIN {X 0,Y 241.703,Z 468.91,A -85,B 0,C 180,E1 -23788.066,E2 -23788.066} C_VEL
LIN {X 0,Y 236.115,Z 484.371,A -85,B 0,C 180,E1 -23789.034,E2 -23789.034} C_VEL
LIN {X 0,Y 229.804,Z 498.879,A -85,B 0,C 180,E1 -23790.239,E2 -23790.239} C_VEL
LIN {X 0,Y 222.26,Z 513.655,A -85,B 0,C 180,E1 -23791.812,E2 -23791.812} C_VEL
LIN {X 0,Y 214.917,Z 526.224,A -85,B 0,C 180,E1 -23793.503,E2 -23793.503} C_VEL
LIN {X 0,Y 207.216,Z 538.083,A -85,B 0,C 180,E1 -23795.514,E2 -23795.514} C_VEL
LIN {X 0,Y 198.619,Z 549.854,A -85,B 0,C 180,E1 -23798.068,E2 -23798.068} C_VEL
LIN {X 0,Y 190.5,Z 559.974,A -85,B 0,C 180,E1 -23800.863,E2 -23800.863} C_VEL
LIN {X 0,Y 182.655,Z 569.028,A -85,B 0,C 180,E1 -23803.982,E2 -23803.982} C_VEL
LIN {X 0,Y 174.001,Z 578.325,A -85,B 0,C 180,E1 -23808.208,E2 -23808.208} C_VEL
LIN {X 0,Y 167.016,Z 585.336,A -85,B 0,C 180,E1 -23812.401,E2 -23812.401} C_VEL
LIN {X 0,Y 161.042,Z 591.229,A -85,B 0,C 180,E1 -23816.942,E2 -23816.942} C_VEL
LIN {X 0,Y 155.079,Z 597.031,A -85,B 0,C 180,E1 -23823.053,E2 -23823.053} C_VEL
LIN {X 0,Y 151.579,Z 600.463,A -85,B 0,C 180,E1 -23828.229,E2 -23828.229} C_VEL
LIN {X 0,Y 149.168,Z 603.016,A -85,B 0,C 180,E1 -23833.58,E2 -23833.58} C_VEL
LIN {X 0,Y 147.886,Z 604.529,A -85,B 0,C 180,E1 -23839.043,E2 -23839.043} C_VEL
LIN {X 0,Y 147.536,Z 605.187,A -85,B 0,C 180,E1 -23844.534,E2 -23844.534} C_VEL
LIN {X 0,Y 147.716,Z 604.796,A -85,B 0,C 180,E1 -23850.001,E2 -23850.001} C_VEL
LIN {X 0,Y 147.641,Z 604.259,A -85,B 0,C 180,E1 -23852.729,E2 -23852.729} C_VEL
LIN {X 0,Y 147.635,Z 602.355,A -85,B 0,C 180,E1 -23858.211,E2 -23858.211} C_VEL
LIN {X 0,Y 148.351,Z 599.411,A -85,B 0,C 180,E1 -23863.703,E2 -23863.703} C_VEL
LIN {X 0,Y 150.142,Z 595.382,A -85,B 0,C 180,E1 -23869.128,E2 -23869.128} C_VEL
LIN {X 0,Y 152.856,Z 590.136,A -85,B 0,C 180,E1 -23874.444,E2 -23874.444} C_VEL
LIN {X 0,Y 156.685,Z 583.684,A -85,B 0,C 180,E1 -23879.564,E2 -23879.564} C_VEL
LIN {X 0,Y 161.592,Z 575.813,A -85,B 0,C 180,E1 -23884.43,E2 -23884.43} C_VEL
LIN {X 0,Y 167.584,Z 566.33,A -85,B 0,C 180,E1 -23888.981,E2 -23888.981} C_VEL
LIN {X 0,Y 173.58,Z 556.526,A -85,B 0,C 180,E1 -23892.702,E2 -23892.702} C_VEL
LIN {X 0,Y 180.221,Z 545.048,A -85,B 0,C 180,E1 -23896.173,E2 -23896.173} C_VEL
LIN {X 0,Y 186.975,Z 532.538,A -85,B 0,C 180,E1 -23899.153,E2 -23899.153} C_VEL
LIN {X 0,Y 193.724,Z 518.759,A -85,B 0,C 180,E1 -23901.711,E2 -23901.711} C_VEL
LIN {X 0,Y 200.12,Z 503.883,A -85,B 0,C 180,E1 -23903.875,E2 -23903.875} C_VEL
LIN {X 0,Y 205.592,Z 489.115,A -85,B 0,C 180,E1 -23905.557,E2 -23905.557} C_VEL
LIN {X 0,Y 210.569,Z 473.04,A -85,B 0,C 180,E1 -23906.99,E2 -23906.99} C_VEL
LIN {X 0,Y 214.73,Z 456.428,A -85,B 0,C 180,E1 -23908.094,E2 -23908.094} C_VEL
LIN {X 0,Y 217.961,Z 440.012,A -85,B 0,C 180,E1 -23908.849,E2 -23908.849} C_VEL
LIN {X 0,Y 220,Z 423.626,A -85,B 0,C 180,E1 -23909.406,E2 -23909.406} C_VEL
LIN {X 0,Y 227.105,Z 342.638,A -85,B 0,C 180,E1 -23911.6,E2 -23911.6} C_VEL
LIN {X 0,Y 221.142,Z 329.071,A -85,B 0,C 180,E1 -23914.668,E2 -23914.668} C_VEL
LIN {X 0,Y 216.765,Z 320.434,A -85,B 0,C 180,E1 -23917.104,E2 -23917.104} C_VEL
LIN {X 0,Y 210.451,Z 310.122,A -85,B 0,C 180,E1 -23920.892,E2 -23920.892} C_VEL
LIN {X 0,Y 205.944,Z 303.266,A -85,B 0,C 180,E1 -23923.966,E2 -23923.966} C_VEL
LIN {X 0,Y 202.612,Z 298.395,A -85,B 0,C 180,E1 -23926.552,E2 -23926.552} C_VEL
LIN {X 0,Y 199.965,Z 294.578,A -85,B 0,C 180,E1 -23928.815,E2 -23928.815} C_VEL
LIN {X 0,Y 197.052,Z 290.438,A -85,B 0,C 180,E1 -23931.659,E2 -23931.659} C_VEL
LIN {X 0,Y 194.36,Z 286.465,A -85,B 0,C 180,E1 -23934.747,E2 -23934.747} C_VEL
LIN {X 0,Y 191.344,Z 282.758,A -85,B 0,C 180,E1 -23938.942,E2 -23938.942} C_VEL
LIN {X 0,Y 190.447,Z 280.834,A -85,B 0,C 180,E1 -23940.661,E2 -23940.661} C_VEL
LIN {X 0,Y 187.818,Z 278.406,A -85,B 0,C 180,E1 -23947.012,E2 -23947.012} C_VEL
LIN {X 0,Y 187.265,Z 276.491,A -85,B 0,C 180,E1 -23950.816,E2 -23950.816} C_VEL
LIN {X 0,Y 187.151,Z 276.412,A -85,B 0,C 180,E1 -23953.751,E2 -23953.751} C_VEL
LIN {X 0,Y 187.583,Z 278.483,A -85,B 0,C 180,E1 -23958.716,E2 -23958.716} C_VEL
LIN {X 0,Y 190.637,Z 281.722,A -85,B 0,C 180,E1 -23966.343,E2 -23966.343} C_VEL
LIN {X 0,Y 192.911,Z 285.388,A -85,B 0,C 180,E1 -23970.011,E2 -23970.011} C_VEL
LIN {X 0,Y 194.338,Z 286.895,A -85,B 0,C 180,E1 -23971.826,E2 -23971.826} C_VEL
LIN {X 0,Y 197.046,Z 290.689,A -85,B 0,C 180,E1 -23974.881,E2 -23974.881} C_VEL
LIN {X 0,Y 198.184,Z 292.309,A -85,B 0,C 180,E1 -23976.054,E2 -23976.054} C_VEL
LIN {X 0,Y 201.324,Z 296.724,A -85,B 0,C 180,E1 -23978.929,E2 -23978.929} C_VEL
LIN {X 0,Y 204.669,Z 301.593,A -85,B 0,C 180,E1 -23981.624,E2 -23981.624} C_VEL
LIN {X 0,Y 207.923,Z 306.342,A -85,B 0,C 180,E1 -23983.962,E2 -23983.962} C_VEL
LIN {X 0,Y 212.603,Z 313.676,A -85,B 0,C 180,E1 -23987.003,E2 -23987.003} C_VEL
LIN {X 0,Y 218.159,Z 322.753,A -85,B 0,C 180,E1 -23990.189,E2 -23990.189} C_VEL
LIN {X 0,Y 224.256,Z 333.768,A -85,B 0,C 180,E1 -23993.351,E2 -23993.351} C_VEL
LIN {X 0,Y 227.142,Z 339.236,A -85,B 0,C 180,E1 -23994.73,E2 -23994.73} C_VEL
LIN {X 0,Y 220.644,Z 413.361,A -85,B 0,C 180,E1 -23996.734,E2 -23996.734} C_VEL
LIN {X 0,Y 218.711,Z 429.815,A -85,B 0,C 180,E1 -23997.277,E2 -23997.277} C_VEL
LIN {X 0,Y 215.749,Z 446.583,A -85,B 0,C 180,E1 -23998.081,E2 -23998.081} C_VEL
LIN {X 0,Y 212.029,Z 462.431,A -85,B 0,C 180,E1 -23999.126,E2 -23999.126} C_VEL
LIN {X 0,Y 207.898,Z 476.814,A -85,B 0,C 180,E1 -24000.37,E2 -24000.37} C_VEL
LIN {X 0,Y 202.645,Z 492.124,A -85,B 0,C 180,E1 -24002.082,E2 -24002.082} C_VEL
LIN {X 0,Y 196.814,Z 506.38,A -85,B 0,C 180,E1 -24004.059,E2 -24004.059} C_VEL
LIN {X 0,Y 190.266,Z 520.669,A -85,B 0,C 180,E1 -24006.604,E2 -24006.604} C_VEL
LIN {X 0,Y 183.926,Z 532.874,A -85,B 0,C 180,E1 -24009.301,E2 -24009.301} C_VEL
LIN {X 0,Y 177.615,Z 544.21,A -85,B 0,C 180,E1 -24012.456,E2 -24012.456} C_VEL
LIN {X 0,Y 170.92,Z 555.223,A -85,B 0,C 180,E1 -24016.323,E2 -24016.323} C_VEL
LIN {X 0,Y 165.33,Z 563.996,A -85,B 0,C 180,E1 -24020.21,E2 -24020.21} C_VEL
LIN {X 0,Y 159.879,Z 572.494,A -85,B 0,C 180,E1 -24024.956,E2 -24024.956} C_VEL
LIN {X 0,Y 155.455,Z 579.549,A -85,B 0,C 180,E1 -24029.999,E2 -24029.999} C_VEL
LIN {X 0,Y 151.933,Z 585.247,A -85,B 0,C 180,E1 -24035.307,E2 -24035.307} C_VEL
LIN {X 0,Y 149.46,Z 589.789,A -85,B 0,C 180,E1 -24040.84,E2 -24040.84} C_VEL
LIN {X 0,Y 147.854,Z 593.233,A -85,B 0,C 180,E1 -24046.57,E2 -24046.57} C_VEL
LIN {X 0,Y 147.118,Z 595.496,A -85,B 0,C 180,E1 -24052.467,E2 -24052.467} C_VEL
LIN {X 0,Y 147.082,Z 596.704,A -85,B 0,C 180,E1 -24058.542,E2 -24058.542} C_VEL
LIN {X 0,Y 147.883,Z 596.76,A -85,B 0,C 180,E1 -24064.769,E2 -24064.769} C_VEL
LIN {X 0,Y 149.848,Z 595.425,A -85,B 0,C 180,E1 -24071.374,E2 -24071.374} C_VEL
LIN {X 0,Y 152.897,Z 592.959,A -85,B 0,C 180,E1 -24077.343,E2 -24077.343} C_VEL
LIN {X 0,Y 157.512,Z 589.009,A -85,B 0,C 180,E1 -24083.429,E2 -24083.429} C_VEL
LIN {X 0,Y 163.663,Z 583.54,A -85,B 0,C 180,E1 -24089.183,E2 -24089.183} C_VEL
LIN {X 0,Y 171.316,Z 576.447,A -85,B 0,C 180,E1 -24094.488,E2 -24094.488} C_VEL
LIN {X 0,Y 179.096,Z 568.7,A -85,B 0,C 180,E1 -24098.743,E2 -24098.743} C_VEL
LIN {X 0,Y 187.649,Z 559.495,A -85,B 0,C 180,E1 -24102.565,E2 -24102.565} C_VEL
LIN {X 0,Y 195.819,Z 549.863,A -85,B 0,C 180,E1 -24105.7,E2 -24105.7} C_VEL
LIN {X 0,Y 204.794,Z 538.287,A -85,B 0,C 180,E1 -24108.597,E2 -24108.597} C_VEL
LIN {X 0,Y 212.653,Z 526.897,A -85,B 0,C 180,E1 -24110.852,E2 -24110.852} C_VEL
LIN {X 0,Y 220.449,Z 514.083,A -85,B 0,C 180,E1 -24112.864,E2 -24112.864} C_VEL
LIN {X 0,Y 227.582,Z 500.791,A -85,B 0,C 180,E1 -24114.529,E2 -24114.529} C_VEL
LIN {X 0,Y 234.009,Z 487.028,A -85,B 0,C 180,E1 -24115.895,E2 -24115.895} C_VEL
LIN {X 0,Y 240.128,Z 471.304,A -85,B 0,C 180,E1 -24117.121,E2 -24117.121} C_VEL
LIN {X 0,Y 244.802,Z 456.36,A -85,B 0,C 180,E1 -24118.027,E2 -24118.027} C_VEL
LIN {X 0,Y 248.869,Z 439.819,A -85,B 0,C 180,E1 -24118.767,E2 -24118.767} C_VEL
LIN {X 0,Y 251.934,Z 422.155,A -85,B 0,C 180,E1 -24119.305,E2 -24119.305} C_VEL
LIN {X 0,Y 259.205,Z 357.461,A -85,B 0,C 180,E1 -24120.832,E2 -24120.832} C_VEL
LIN {X 0,Y 257.45,Z 353.153,A -85,B 0,C 180,E1 -24122.949,E2 -24122.949} C_VEL
LIN {X 0,Y 255.708,Z 348.823,A -85,B 0,C 180,E1 -24125.738,E2 -24125.738} C_VEL
LIN {X 0,Y 255.074,Z 347.463,A -85,B 0,C 180,E1 -24127.045,E2 -24127.045} C_VEL
LIN {X 0,Y 253.964,Z 344.68,A -85,B 0,C 180,E1 -24131.169,E2 -24131.169} C_VEL
LIN {X 0,Y 253.955,Z 343.904,A -85,B 0,C 180,E1 -24132.077,E2 -24132.077} C_VEL
LIN {X 0,Y 253.918,Z 343.942,A -85,B 0,C 180,E1 -24133.046,E2 -24133.046} C_VEL
LIN {X 0,Y 255.104,Z 347.981,A -85,B 0,C 180,E1 -24138.765,E2 -24138.765} C_VEL
LIN {X 0,Y 256.555,Z 351.4,A -85,B 0,C 180,E1 -24141.418,E2 -24141.418} C_VEL
LIN {X 0,Y 257.891,Z 354.644,A -85,B 0,C 180,E1 -24143.291,E2 -24143.291} C_VEL
LIN {X 0,Y 259.128,Z 358.576,A -85,B 0,C 180,E1 -24144.857,E2 -24144.857} C_VEL
LIN {X 0,Y 251.018,Z 430.265,A -85,B 0,C 180,E1 -24146.567,E2 -24146.567} C_VEL
LIN {X 0,Y 247.722,Z 447.43,A -85,B 0,C 180,E1 -24147.11,E2 -24147.11} C_VEL
LIN {X 0,Y 243.3,Z 463.825,A -85,B 0,C 180,E1 -24147.796,E2 -24147.796} C_VEL
LIN {X 0,Y 241.703,Z 468.91,A -85,B 0,C 180,E1 -24148.066,E2 -24148.066} C_VEL
LIN {X 0,Y 239.615,Z 474.525,A -85,B 0,C 180,E1 -24148.246,E2 -24148.246} C_VEL
LIN {X 0,Y 235.215,Z 483.542,A -85,B 0,C 180,E1 -24148.155,E2 -24148.155} C_VEL
LIN {X 0,Y 230.572,Z 492.14,A -85,B 0,C 180,E1 -24148.119,E2 -24148.119} C_VEL
LIN {X 0,Y 227.972,Z 497.202,A -85,B 0,C 180,E1 -24148.398,E2 -24148.398} C_VEL
LIN {X 0,Y 220.765,Z 511.323,A -85,B 0,C 180,E1 -24149.833,E2 -24149.833} C_VEL
LIN {X 0,Y 213.146,Z 524.233,A -85,B 0,C 180,E1 -24151.444,E2 -24151.444} C_VEL
LIN {X 0,Y 204.493,Z 537.218,A -85,B 0,C 180,E1 -24153.59,E2 -24153.59} C_VEL
LIN {X 0,Y 195.592,Z 549.008,A -85,B 0,C 180,E1 -24156.056,E2 -24156.056} C_VEL
LIN {X 0,Y 187.118,Z 559.236,A -85,B 0,C 180,E1 -24158.801,E2 -24158.801} C_VEL
LIN {X 0,Y 178.655,Z 568.57,A -85,B 0,C 180,E1 -24161.971,E2 -24161.971} C_VEL
LIN {X 0,Y 170.701,Z 576.665,A -85,B 0,C 180,E1 -24165.582,E2 -24165.582} C_VEL
LIN {X 0,Y 163.142,Z 583.96,A -85,B 0,C 180,E1 -24169.747,E2 -24169.747} C_VEL
LIN {X 0,Y 156.525,Z 590.015,A -85,B 0,C 180,E1 -24174.29,E2 -24174.29} C_VEL
LIN {X 0,Y 151.016,Z 594.94,A -85,B 0,C 180,E1 -24179.21,E2 -24179.21} C_VEL
LIN {X 0,Y 146.643,Z 598.877,A -85,B 0,C 180,E1 -24184.449,E2 -24184.449} C_VEL
LIN {X 0,Y 143.456,Z 601.781,A -85,B 0,C 180,E1 -24189.945,E2 -24189.945} C_VEL
LIN {X 0,Y 141.392,Z 603.766,A -85,B 0,C 180,E1 -24195.611,E2 -24195.611} C_VEL
LIN {X 0,Y 140.526,Z 604.784,A -85,B 0,C 180,E1 -24201.372,E2 -24201.372} C_VEL
LIN {X 0,Y 140.5,Z 604.875,A -85,B 0,C 180,E1 -24207.134,E2 -24207.134} C_VEL
LIN {X 0,Y 140.578,Z 604.386,A -85,B 0,C 180,E1 -24210.936,E2 -24210.936} C_VEL
LIN {X 0,Y 140.491,Z 603.15,A -85,B 0,C 180,E1 -24215.743,E2 -24215.743} C_VEL
LIN {X 0,Y 140.846,Z 600.63,A -85,B 0,C 180,E1 -24221.514,E2 -24221.514} C_VEL
LIN {X 0,Y 142.273,Z 597.109,A -85,B 0,C 180,E1 -24227.241,E2 -24227.241} C_VEL
LIN {X 0,Y 144.667,Z 592.4,A -85,B 0,C 180,E1 -24232.871,E2 -24232.871} C_VEL
LIN {X 0,Y 148.219,Z 586.479,A -85,B 0,C 180,E1 -24238.305,E2 -24238.305} C_VEL
LIN {X 0,Y 152.913,Z 579.272,A -85,B 0,C 180,E1 -24243.472,E2 -24243.472} C_VEL
LIN {X 0,Y 158.716,Z 570.54,A -85,B 0,C 180,E1 -24248.311,E2 -24248.311} C_VEL
LIN {X 0,Y 164.703,Z 561.466,A -85,B 0,C 180,E1 -24252.227,E2 -24252.227} C_VEL
LIN {X 0,Y 171.229,Z 550.872,A -85,B 0,C 180,E1 -24255.911,E2 -24255.911} C_VEL
LIN {X 0,Y 177.395,Z 540.337,A -85,B 0,C 180,E1 -24258.828,E2 -24258.828} C_VEL
LIN {X 0,Y 184.058,Z 528.045,A -85,B 0,C 180,E1 -24261.514,E2 -24261.514} C_VEL
LIN {X 0,Y 190.263,Z 515.244,A -85,B 0,C 180,E1 -24263.771,E2 -24263.771} C_VEL
LIN {X 0,Y 196.566,Z 500.725,A -85,B 0,C 180,E1 -24265.772,E2 -24265.772} C_VEL
LIN {X 0,Y 202.213,Z 485.393,A -85,B 0,C 180,E1 -24267.439,E2 -24267.439} C_VEL
LIN {X 0,Y 207.359,Z 468.375,A -85,B 0,C 180,E1 -24268.848,E2 -24268.848} C_VEL
LIN {X 0,Y 211.393,Z 451.841,A -85,B 0,C 180,E1 -24269.814,E2 -24269.814} C_VEL
LIN {X 0,Y 214.347,Z 435.513,A -85,B 0,C 180,E1 -24270.491,E2 -24270.491} C_VEL
LIN {X 0,Y 216.693,Z 412.938,A -85,B 0,C 180,E1 -24271.197,E2 -24271.197} C_VEL
LIN {X 0,Y 222.801,Z 345.493,A -85,B 0,C 180,E1 -24273.003,E2 -24273.003} C_VEL
LIN {X 0,Y 217.451,Z 333.133,A -85,B 0,C 180,E1 -24275.934,E2 -24275.934} C_VEL
LIN {X 0,Y 213.952,Z 326.125,A -85,B 0,C 180,E1 -24277.968,E2 -24277.968} C_VEL
LIN {X 0,Y 208.273,Z 316.485,A -85,B 0,C 180,E1 -24281.548,E2 -24281.548} C_VEL
LIN {X 0,Y 203.927,Z 309.672,A -85,B 0,C 180,E1 -24284.622,E2 -24284.622} C_VEL
LIN {X 0,Y 200.719,Z 304.845,A -85,B 0,C 180,E1 -24287.206,E2 -24287.206} C_VEL
LIN {X 0,Y 197.978,Z 300.789,A -85,B 0,C 180,E1 -24289.662,E2 -24289.662} C_VEL
LIN {X 0,Y 195.542,Z 297.159,A -85,B 0,C 180,E1 -24292.165,E2 -24292.165} C_VEL
LIN {X 0,Y 192.854,Z 293.073,A -85,B 0,C 180,E1 -24295.372,E2 -24295.372} C_VEL
LIN {X 0,Y 190.103,Z 289.631,A -85,B 0,C 180,E1 -24299.355,E2 -24299.355} C_VEL
LIN {X 0,Y 189.256,Z 287.746,A -85,B 0,C 180,E1 -24301.064,E2 -24301.064} C_VEL
LIN {X 0,Y 186.807,Z 285.411,A -85,B 0,C 180,E1 -24307.24,E2 -24307.24} C_VEL
LIN {X 0,Y 186.282,Z 283.463,A -85,B 0,C 180,E1 -24311.211,E2 -24311.211} C_VEL
LIN {X 0,Y 186.198,Z 283.523,A -85,B 0,C 180,E1 -24313.823,E2 -24313.823} C_VEL
LIN {X 0,Y 186.576,Z 285.452,A -85,B 0,C 180,E1 -24318.455,E2 -24318.455} C_VEL
LIN {X 0,Y 189.373,Z 288.512,A -85,B 0,C 180,E1 -24325.816,E2 -24325.816} C_VEL
LIN {X 0,Y 191.616,Z 292.223,A -85,B 0,C 180,E1 -24329.588,E2 -24329.588} C_VEL
LIN {X 0,Y 192.847,Z 293.549,A -85,B 0,C 180,E1 -24331.222,E2 -24331.222} C_VEL
LIN {X 0,Y 195.711,Z 297.602,A -85,B 0,C 180,E1 -24334.574,E2 -24334.574} C_VEL
LIN {X 0,Y 199.51,Z 303.257,A -85,B 0,C 180,E1 -24338.305,E2 -24338.305} C_VEL
LIN {X 0,Y 202.529,Z 307.723,A -85,B 0,C 180,E1 -24340.822,E2 -24340.822} C_VEL
LIN {X 0,Y 206.66,Z 313.922,A -85,B 0,C 180,E1 -24343.889,E2 -24343.889} C_VEL
LIN {X 0,Y 212.947,Z 324.322,A -85,B 0,C 180,E1 -24347.957,E2 -24347.957} C_VEL
LIN {X 0,Y 218.276,Z 333.783,A -85,B 0,C 180,E1 -24350.977,E2 -24350.977} C_VEL
LIN {X 0,Y 222.809,Z 342.497,A -85,B 0,C 180,E1 -24353.336,E2 -24353.336} C_VEL
LIN {X 0,Y 215.357,Z 423.435,A -85,B 0,C 180,E1 -24355.552,E2 -24355.552} C_VEL
LIN {X 0,Y 212.693,Z 440.193,A -85,B 0,C 180,E1 -24356.238,E2 -24356.238} C_VEL
LIN {X 0,Y 209.207,Z 456.271,A -85,B 0,C 180,E1 -24357.184,E2 -24357.184} C_VEL
LIN {X 0,Y 204.791,Z 472.279,A -85,B 0,C 180,E1 -24358.443,E2 -24358.443} C_VEL
LIN {X 0,Y 199.886,Z 486.98,A -85,B 0,C 180,E1 -24359.932,E2 -24359.932} C_VEL
LIN {X 0,Y 193.857,Z 502.167,A -85,B 0,C 180,E1 -24361.881,E2 -24361.881} C_VEL
LIN {X 0,Y 187.978,Z 515.076,A -85,B 0,C 180,E1 -24364.003,E2 -24364.003} C_VEL
LIN {X 0,Y 181.4,Z 527.886,A -85,B 0,C 180,E1 -24366.602,E2 -24366.602} C_VEL
LIN {X 0,Y 175.136,Z 539.096,A -85,B 0,C 180,E1 -24369.443,E2 -24369.443} C_VEL
LIN {X 0,Y 168.362,Z 550.265,A -85,B 0,C 180,E1 -24373.01,E2 -24373.01} C_VEL
LIN {X 0,Y 161.325,Z 561.043,A -85,B 0,C 180,E1 -24377.418,E2 -24377.418} C_VEL
LIN {X 0,Y 155.273,Z 570.033,A -85,B 0,C 180,E1 -24382.195,E2 -24382.195} C_VEL
LIN {X 0,Y 150.217,Z 577.525,A -85,B 0,C 180,E1 -24387.318,E2 -24387.318} C_VEL
LIN {X 0,Y 146.2,Z 583.714,A -85,B 0,C 180,E1 -24392.755,E2 -24392.755} C_VEL
LIN {X 0,Y 143.217,Z 588.622,A -85,B 0,C 180,E1 -24398.465,E2 -24398.465} C_VEL
LIN {X 0,Y 141.19,Z 592.396,A -85,B 0,C 180,E1 -24404.41,E2 -24404.41} C_VEL
LIN {X 0,Y 140.127,Z 595.11,A -85,B 0,C 180,E1 -24410.552,E2 -24410.552} C_VEL
LIN {X 0,Y 139.928,Z 596.359,A -85,B 0,C 180,E1 -24415.302,E2 -24415.302} C_VEL
LIN {X 0,Y 140.277,Z 597.095,A -85,B 0,C 180,E1 -24421.601,E2 -24421.601} C_VEL
LIN {X 0,Y 141.32,Z 596.741,A -85,B 0,C 180,E1 -24427.279,E2 -24427.279} C_VEL
LIN {X 0,Y 143.493,Z 595.429,A -85,B 0,C 180,E1 -24433.288,E2 -24433.288} C_VEL
LIN {X 0,Y 147.243,Z 592.624,A -85,B 0,C 180,E1 -24439.788,E2 -24439.788} C_VEL
LIN {X 0,Y 153.063,Z 587.978,A -85,B 0,C 180,E1 -24446.565,E2 -24446.565} C_VEL
LIN {X 0,Y 159.413,Z 582.681,A -85,B 0,C 180,E1 -24451.849,E2 -24451.849} C_VEL
LIN {X 0,Y 166.661,Z 576.34,A -85,B 0,C 180,E1 -24456.514,E2 -24456.514} C_VEL
LIN {X 0,Y 174.348,Z 569.106,A -85,B 0,C 180,E1 -24460.505,E2 -24460.505} C_VEL
LIN {X 0,Y 182.691,Z 560.625,A -85,B 0,C 180,E1 -24464.093,E2 -24464.093} C_VEL
LIN {X 0,Y 191.267,Z 551.063,A -85,B 0,C 180,E1 -24467.264,E2 -24467.264} C_VEL
LIN {X 0,Y 200.601,Z 539.572,A -85,B 0,C 180,E1 -24470.172,E2 -24470.172} C_VEL
LIN {X 0,Y 209.783,Z 526.78,A -85,B 0,C 180,E1 -24472.682,E2 -24472.682} C_VEL
LIN {X 0,Y 218.077,Z 513.573,A -85,B 0,C 180,E1 -24474.688,E2 -24474.688} C_VEL
LIN {X 0,Y 225.36,Z 500.223,A -85,B 0,C 180,E1 -24476.301,E2 -24476.301} C_VEL
LIN {X 0,Y 232.613,Z 484.736,A -85,B 0,C 180,E1 -24477.744,E2 -24477.744} C_VEL
LIN {X 0,Y 238.402,Z 469.872,A -85,B 0,C 180,E1 -24478.854,E2 -24478.854} C_VEL
LIN {X 0,Y 243.421,Z 453.964,A -85,B 0,C 180,E1 -24479.76,E2 -24479.76} C_VEL
LIN {X 0,Y 247.519,Z 436.9,A -85,B 0,C 180,E1 -24480.444,E2 -24480.444} C_VEL
LIN {X 0,Y 250.289,Z 420.09,A -85,B 0,C 180,E1 -24480.918,E2 -24480.918} C_VEL
LIN {X 0,Y 256.953,Z 361.953,A -85,B 0,C 180,E1 -24482.258,E2 -24482.258} C_VEL
LIN {X 0,Y 255.501,Z 358.478,A -85,B 0,C 180,E1 -24484.3,E2 -24484.3} C_VEL
LIN {X 0,Y 254.405,Z 355.335,A -85,B 0,C 180,E1 -24486.344,E2 -24486.344} C_VEL
LIN {X 0,Y 253.917,Z 354.325,A -85,B 0,C 180,E1 -24487.457,E2 -24487.457} C_VEL
LIN {X 0,Y 252.979,Z 351.297,A -85,B 0,C 180,E1 -24491.82,E2 -24491.82} C_VEL
LIN {X 0,Y 252.964,Z 350.919,A -85,B 0,C 180,E1 -24492.842,E2 -24492.842} C_VEL
LIN {X 0,Y 254.021,Z 354.948,A -85,B 0,C 180,E1 -24498.525,E2 -24498.525} C_VEL
LIN {X 0,Y 255.267,Z 358.102,A -85,B 0,C 180,E1 -24500.972,E2 -24500.972} C_VEL
LIN {X 0,Y 256.449,Z 361.273,A -85,B 0,C 180,E1 -24502.795,E2 -24502.795} C_VEL
LIN {X 0,Y 256.905,Z 362.886,A -85,B 0,C 180,E1 -24503.438,E2 -24503.438} C_VEL
LIN {X 0,Y 249.089,Z 429.902,A -85,B 0,C 180,E1 -24504.991,E2 -24504.991} C_VEL
LIN {X 0,Y 245.829,Z 446.542,A -85,B 0,C 180,E1 -24505.5,E2 -24505.5} C_VEL
LIN {X 0,Y 241.267,Z 463.217,A -85,B 0,C 180,E1 -24506.164,E2 -24506.164} C_VEL
LIN {X 0,Y 235.727,Z 479.123,A -85,B 0,C 180,E1 -24507.041,E2 -24507.041} C_VEL
LIN {X 0,Y 229.206,Z 494.576,A -85,B 0,C 180,E1 -24508.173,E2 -24508.173} C_VEL
LIN {X 0,Y 227.972,Z 497.202,A -85,B 0,C 180,E1 -24508.398,E2 -24508.398} C_VEL
LIN {X 0,Y 225.296,Z 502.33,A -85,B 0,C 180,E1 -24508.719,E2 -24508.719} C_VEL
LIN {X 0,Y 219.945,Z 510.644,A -85,B 0,C 180,E1 -24508.883,E2 -24508.883} C_VEL
LIN {X 0,Y 214.217,Z 518.681,A -85,B 0,C 180,E1 -24509.104,E2 -24509.104} C_VEL
LIN {X 0,Y 210.967,Z 523.34,A -85,B 0,C 180,E1 -24509.535,E2 -24509.535} C_VEL
LIN {X 0,Y 201.952,Z 536.462,A -85,B 0,C 180,E1 -24511.597,E2 -24511.597} C_VEL
LIN {X 0,Y 192.799,Z 548.232,A -85,B 0,C 180,E1 -24513.976,E2 -24513.976} C_VEL
LIN {X 0,Y 183.969,Z 558.51,A -85,B 0,C 180,E1 -24516.657,E2 -24516.657} C_VEL
LIN {X 0,Y 174.438,Z 568.599,A -85,B 0,C 180,E1 -24520.051,E2 -24520.051} C_VEL
LIN {X 0,Y 165.677,Z 577.058,A -85,B 0,C 180,E1 -24523.853,E2 -24523.853} C_VEL
LIN {X 0,Y 157.753,Z 584.203,A -85,B 0,C 180,E1 -24528.069,E2 -24528.069} C_VEL
LIN {X 0,Y 150.76,Z 590.198,A -85,B 0,C 180,E1 -24532.699,E2 -24532.699} C_VEL
LIN {X 0,Y 143.618,Z 596.101,A -85,B 0,C 180,E1 -24539.083,E2 -24539.083} C_VEL
LIN {X 0,Y 140.191,Z 598.904,A -85,B 0,C 180,E1 -24543.182,E2 -24543.182} C_VEL
LIN {X 0,Y 136.737,Z 601.713,A -85,B 0,C 180,E1 -24548.914,E2 -24548.914} C_VEL
LIN {X 0,Y 134.451,Z 603.658,A -85,B 0,C 180,E1 -24554.85,E2 -24554.85} C_VEL
LIN {X 0,Y 133.47,Z 604.595,A -85,B 0,C 180,E1 -24560.912,E2 -24560.912} C_VEL
LIN {X 0,Y 133.399,Z 604.649,A -85,B 0,C 180,E1 -24566.981,E2 -24566.981} C_VEL
LIN {X 0,Y 133.531,Z 604.272,A -85,B 0,C 180,E1 -24570.001,E2 -24570.001} C_VEL
LIN {X 0,Y 133.459,Z 603.661,A -85,B 0,C 180,E1 -24573.019,E2 -24573.019} C_VEL
LIN {X 0,Y 133.507,Z 601.68,A -85,B 0,C 180,E1 -24579.087,E2 -24579.087} C_VEL
LIN {X 0,Y 134.443,Z 598.576,A -85,B 0,C 180,E1 -24585.152,E2 -24585.152} C_VEL
LIN {X 0,Y 136.633,Z 594.45,A -85,B 0,C 180,E1 -24591.105,E2 -24591.105} C_VEL
LIN {X 0,Y 140.817,Z 587.537,A -85,B 0,C 180,E1 -24598.304,E2 -24598.304} C_VEL
LIN {X 0,Y 145.549,Z 580.531,A -85,B 0,C 180,E1 -24603.731,E2 -24603.731} C_VEL
LIN {X 0,Y 151.467,Z 572.072,A -85,B 0,C 180,E1 -24608.785,E2 -24608.785} C_VEL
LIN {X 0,Y 158.477,Z 561.963,A -85,B 0,C 180,E1 -24613.423,E2 -24613.423} C_VEL
LIN {X 0,Y 165.122,Z 551.66,A -85,B 0,C 180,E1 -24617.149,E2 -24617.149} C_VEL
LIN {X 0,Y 172.715,Z 539.181,A -85,B 0,C 180,E1 -24620.636,E2 -24620.636} C_VEL
LIN {X 0,Y 180.232,Z 525.625,A -85,B 0,C 180,E1 -24623.538,E2 -24623.538} C_VEL
LIN {X 0,Y 187.53,Z 510.669,A -85,B 0,C 180,E1 -24626.014,E2 -24626.014} C_VEL
LIN {X 0,Y 193.845,Z 495.631,A -85,B 0,C 180,E1 -24627.938,E2 -24627.938} C_VEL
LIN {X 0,Y 199.053,Z 481.109,A -85,B 0,C 180,E1 -24629.385,E2 -24629.385} C_VEL
LIN {X 0,Y 203.719,Z 465.527,A -85,B 0,C 180,E1 -24630.585,E2 -24630.585} C_VEL
LIN {X 0,Y 207.684,Z 449.122,A -85,B 0,C 180,E1 -24631.495,E2 -24631.495} C_VEL
LIN {X 0,Y 210.735,Z 431.397,A -85,B 0,C 180,E1 -24632.185,E2 -24632.185} C_VEL
LIN {X 0,Y 218.602,Z 348.435,A -85,B 0,C 180,E1 -24634.449,E2 -24634.449} C_VEL
LIN {X 0,Y 213.683,Z 336.821,A -85,B 0,C 180,E1 -24637.334,E2 -24637.334} C_VEL
LIN {X 0,Y 211.028,Z 331.474,A -85,B 0,C 180,E1 -24638.958,E2 -24638.958} C_VEL
LIN {X 0,Y 205.705,Z 322.227,A -85,B 0,C 180,E1 -24642.477,E2 -24642.477} C_VEL
LIN {X 0,Y 201.829,Z 315.905,A -85,B 0,C 180,E1 -24645.377,E2 -24645.377} C_VEL
LIN {X 0,Y 198.424,Z 310.69,A -85,B 0,C 180,E1 -24648.236,E2 -24648.236} C_VEL
LIN {X 0,Y 196.3,Z 307.383,A -85,B 0,C 180,E1 -24650.259,E2 -24650.259} C_VEL
LIN {X 0,Y 193.852,Z 303.684,A -85,B 0,C 180,E1 -24652.862,E2 -24652.862} C_VEL
LIN {X 0,Y 191.224,Z 299.572,A -85,B 0,C 180,E1 -24656.199,E2 -24656.199} C_VEL
LIN {X 0,Y 188.685,Z 296.128,A -85,B 0,C 180,E1 -24660.137,E2 -24660.137} C_VEL
LIN {X 0,Y 187.999,Z 294.607,A -85,B 0,C 180,E1 -24661.619,E2 -24661.619} C_VEL
LIN {X 0,Y 185.77,Z 292.319,A -85,B 0,C 180,E1 -24667.636,E2 -24667.636} C_VEL
LIN {X 0,Y 185.345,Z 290.621,A -85,B 0,C 180,E1 -24670.929,E2 -24670.929} C_VEL
LIN {X 0,Y 185.258,Z 290.408,A -85,B 0,C 180,E1 -24673.157,E2 -24673.157} C_VEL
LIN {X 0,Y 185.347,Z 291.7,A -85,B 0,C 180,E1 -24676.649,E2 -24676.649} C_VEL
LIN {X 0,Y 188.175,Z 295.457,A -85,B 0,C 180,E1 -24685.405,E2 -24685.405} C_VEL
LIN {X 0,Y 190.502,Z 299.234,A -85,B 0,C 180,E1 -24689.42,E2 -24689.42} C_VEL
LIN {X 0,Y 191.528,Z 300.499,A -85,B 0,C 180,E1 -24690.829,E2 -24690.829} C_VEL
LIN {X 0,Y 194.749,Z 305.292,A -85,B 0,C 180,E1 -24694.687,E2 -24694.687} C_VEL
LIN {X 0,Y 197.63,Z 309.629,A -85,B 0,C 180,E1 -24697.582,E2 -24697.582} C_VEL
LIN {X 0,Y 201.169,Z 315.056,A -85,B 0,C 180,E1 -24700.627,E2 -24700.627} C_VEL
LIN {X 0,Y 205.062,Z 321.236,A -85,B 0,C 180,E1 -24703.602,E2 -24703.602} C_VEL
LIN {X 0,Y 210.639,Z 330.679,A -85,B 0,C 180,E1 -24707.314,E2 -24707.314} C_VEL
LIN {X 0,Y 216.179,Z 340.925,A -85,B 0,C 180,E1 -24710.563,E2 -24710.563} C_VEL
LIN {X 0,Y 218.577,Z 345.672,A -85,B 0,C 180,E1 -24711.878,E2 -24711.878} C_VEL
LIN {X 0,Y 212.269,Z 413.678,A -85,B 0,C 180,E1 -24713.713,E2 -24713.713} C_VEL
LIN {X 0,Y 210.168,Z 430.473,A -85,B 0,C 180,E1 -24714.257,E2 -24714.257} C_VEL
LIN {X 0,Y 206.966,Z 447.516,A -85,B 0,C 180,E1 -24715.068,E2 -24715.068} C_VEL
LIN {X 0,Y 203,Z 463.423,A -85,B 0,C 180,E1 -24716.122,E2 -24716.122} C_VEL
LIN {X 0,Y 198.667,Z 477.65,A -85,B 0,C 180,E1 -24717.352,E2 -24717.352} C_VEL
LIN {X 0,Y 193.086,Z 492.9,A -85,B 0,C 180,E1 -24719.061,E2 -24719.061} C_VEL
LIN {X 0,Y 186.904,Z 507.094,A -85,B 0,C 180,E1 -24721.044,E2 -24721.044} C_VEL
LIN {X 0,Y 180.12,Z 520.96,A -85,B 0,C 180,E1 -24723.542,E2 -24723.542} C_VEL
LIN {X 0,Y 173.649,Z 532.61,A -85,B 0,C 180,E1 -24726.126,E2 -24726.126} C_VEL
LIN {X 0,Y 166.323,Z 544.8,A -85,B 0,C 180,E1 -24729.598,E2 -24729.598} C_VEL
LIN {X 0,Y 159.506,Z 555.134,A -85,B 0,C 180,E1 -24733.357,E2 -24733.357} C_VEL
LIN {X 0,Y 153.37,Z 563.998,A -85,B 0,C 180,E1 -24737.428,E2 -24737.428} C_VEL
LIN {X 0,Y 148.002,Z 571.616,A -85,B 0,C 180,E1 -24741.809,E2 -24741.809} C_VEL
LIN {X 0,Y 142.884,Z 578.837,A -85,B 0,C 180,E1 -24747.18,E2 -24747.18} C_VEL
LIN {X 0,Y 138.795,Z 584.785,A -85,B 0,C 180,E1 -24752.902,E2 -24752.902} C_VEL
LIN {X 0,Y 135.857,Z 589.562,A -85,B 0,C 180,E1 -24758.927,E2 -24758.927} C_VEL
LIN {X 0,Y 133.883,Z 593.122,A -85,B 0,C 180,E1 -24765.215,E2 -24765.215} C_VEL
LIN {X 0,Y 132.938,Z 595.615,A -85,B 0,C 180,E1 -24771.719,E2 -24771.719} C_VEL
LIN {X 0,Y 132.839,Z 596.615,A -85,B 0,C 180,E1 -24775.92,E2 -24775.92} C_VEL
LIN {X 0,Y 133.284,Z 597.319,A -85,B 0,C 180,E1 -24782.47,E2 -24782.47} C_VEL
LIN {X 0,Y 134.61,Z 596.88,A -85,B 0,C 180,E1 -24788.792,E2 -24788.792} C_VEL
LIN {X 0,Y 137.442,Z 595.24,A -85,B 0,C 180,E1 -24795.713,E2 -24795.713} C_VEL
LIN {X 0,Y 141.847,Z 592.277,A -85,B 0,C 180,E1 -24802.44,E2 -24802.44} C_VEL
LIN {X 0,Y 147.851,Z 587.823,A -85,B 0,C 180,E1 -24808.825,E2 -24808.825} C_VEL
LIN {X 0,Y 155.542,Z 581.828,A -85,B 0,C 180,E1 -24814.642,E2 -24814.642} C_VEL
LIN {X 0,Y 163.426,Z 575.223,A -85,B 0,C 180,E1 -24819.279,E2 -24819.279} C_VEL
LIN {X 0,Y 172.117,Z 567.377,A -85,B 0,C 180,E1 -24823.392,E2 -24823.392} C_VEL
LIN {X 0,Y 180.537,Z 559.054,A -85,B 0,C 180,E1 -24826.701,E2 -24826.701} C_VEL
LIN {X 0,Y 189.77,Z 548.956,A -85,B 0,C 180,E1 -24829.819,E2 -24829.819} C_VEL
LIN {X 0,Y 199.333,Z 537.326,A -85,B 0,C 180,E1 -24832.566,E2 -24832.566} C_VEL
LIN {X 0,Y 207.847,Z 525.646,A -85,B 0,C 180,E1 -24834.735,E2 -24834.735} C_VEL
LIN {X 0,Y 216.28,Z 512.468,A -85,B 0,C 180,E1 -24836.644,E2 -24836.644} C_VEL
LIN {X 0,Y 223.924,Z 498.68,A -85,B 0,C 180,E1 -24838.201,E2 -24838.201} C_VEL
LIN {X 0,Y 230.611,Z 484.583,A -85,B 0,C 180,E1 -24839.465,E2 -24839.465} C_VEL
LIN {X 0,Y 236.52,Z 469.733,A -85,B 0,C 180,E1 -24840.524,E2 -24840.524} C_VEL
LIN {X 0,Y 241.436,Z 454.487,A -85,B 0,C 180,E1 -24841.361,E2 -24841.361} C_VEL
LIN {X 0,Y 245.449,Z 438.277,A -85,B 0,C 180,E1 -24842,E2 -24842} C_VEL
LIN {X 0,Y 248.36,Z 421.547,A -85,B 0,C 180,E1 -24842.469,E2 -24842.469} C_VEL
LIN {X 0,Y 254.876,Z 366.729,A -85,B 0,C 180,E1 -24843.707,E2 -24843.707} C_VEL
LIN {X 0,Y 253.186,Z 361.927,A -85,B 0,C 180,E1 -24846.891,E2 -24846.891} C_VEL
LIN {X 0,Y 252.013,Z 357.976,A -85,B 0,C 180,E1 -24852.568,E2 -24852.568} C_VEL
LIN {X 0,Y 252.887,Z 361.728,A -85,B 0,C 180,E1 -24858.124,E2 -24858.124} C_VEL
LIN {X 0,Y 254.104,Z 365.054,A -85,B 0,C 180,E1 -24860.709,E2 -24860.709} C_VEL
LIN {X 0,Y 254.866,Z 367.203,A -85,B 0,C 180,E1 -24861.98,E2 -24861.98} C_VEL
LIN {X 0,Y 247.339,Z 429.775,A -85,B 0,C 180,E1 -24863.4,E2 -24863.4} C_VEL
LIN {X 0,Y 244.004,Z 446.447,A -85,B 0,C 180,E1 -24863.893,E2 -24863.893} C_VEL
LIN {X 0,Y 239.447,Z 462.797,A -85,B 0,C 180,E1 -24864.514,E2 -24864.514} C_VEL
LIN {X 0,Y 234.191,Z 477.785,A -85,B 0,C 180,E1 -24865.308,E2 -24865.308} C_VEL
LIN {X 0,Y 228.237,Z 491.89,A -85,B 0,C 180,E1 -24866.258,E2 -24866.258} C_VEL
LIN {X 0,Y 221.705,Z 505.008,A -85,B 0,C 180,E1 -24867.43,E2 -24867.43} C_VEL
LIN {X 0,Y 213.845,Z 518.718,A -85,B 0,C 180,E1 -24868.954,E2 -24868.954} C_VEL
LIN {X 0,Y 210.967,Z 523.34,A -85,B 0,C 180,E1 -24869.535,E2 -24869.535} C_VEL
LIN {X 0,Y 207.641,Z 527.951,A -85,B 0,C 180,E1 -24870.019,E2 -24870.019} C_VEL
LIN {X 0,Y 196.055,Z 541.102,A -85,B 0,C 180,E1 -24870.89,E2 -24870.89} C_VEL
LIN {X 0,Y 192.252,Z 545.259,A -85,B 0,C 180,E1 -24871.414,E2 -24871.414} C_VEL
LIN {X 0,Y 191.066,Z 546.579,A -85,B 0,C 180,E1 -24871.659,E2 -24871.659} C_VEL
LIN {X 0,Y 181.098,Z 557.853,A -85,B 0,C 180,E1 -24874.448,E2 -24874.448} C_VEL
LIN {X 0,Y 171.147,Z 567.959,A -85,B 0,C 180,E1 -24877.771,E2 -24877.771} C_VEL
LIN {X 0,Y 160.815,Z 577.453,A -85,B 0,C 180,E1 -24882.02,E2 -24882.02} C_VEL
LIN {X 0,Y 152.488,Z 584.479,A -85,B 0,C 180,E1 -24886.266,E2 -24886.266} C_VEL
LIN {X 0,Y 145.118,Z 590.386,A -85,B 0,C 180,E1 -24890.982,E2 -24890.982} C_VEL
LIN {X 0,Y 137.486,Z 596.187,A -85,B 0,C 180,E1 -24897.54,E2 -24897.54} C_VEL
LIN {X 0,Y 131.804,Z 600.406,A -85,B 0,C 180,E1 -24904.751,E2 -24904.751} C_VEL
LIN {X 0,Y 128.658,Z 602.703,A -85,B 0,C 180,E1 -24910.869,E2 -24910.869} C_VEL
LIN {X 0,Y 126.837,Z 604.081,A -85,B 0,C 180,E1 -24917.196,E2 -24917.196} C_VEL
LIN {X 0,Y 126.243,Z 604.528,A -85,B 0,C 180,E1 -24923.608,E2 -24923.608} C_VEL
LIN {X 0,Y 126.297,Z 604.422,A -85,B 0,C 180,E1 -24926.811,E2 -24926.811} C_VEL
LIN {X 0,Y 126.444,Z 604.006,A -85,B 0,C 180,E1 -24930.001,E2 -24930.001} C_VEL
LIN {X 0,Y 126.367,Z 603.353,A -85,B 0,C 180,E1 -24933.189,E2 -24933.189} C_VEL
LIN {X 0,Y 126.462,Z 601.326,A -85,B 0,C 180,E1 -24939.598,E2 -24939.598} C_VEL
LIN {X 0,Y 127.529,Z 598.138,A -85,B 0,C 180,E1 -24945.995,E2 -24945.995} C_VEL
LIN {X 0,Y 129.913,Z 593.919,A -85,B 0,C 180,E1 -24952.253,E2 -24952.253} C_VEL
LIN {X 0,Y 133.415,Z 588.46,A -85,B 0,C 180,E1 -24958.301,E2 -24958.301} C_VEL
LIN {X 0,Y 138.21,Z 581.713,A -85,B 0,C 180,E1 -24964.012,E2 -24964.012} C_VEL
LIN {X 0,Y 144.203,Z 573.573,A -85,B 0,C 180,E1 -24969.315,E2 -24969.315} C_VEL
LIN {X 0,Y 151.347,Z 563.821,A -85,B 0,C 180,E1 -24974.151,E2 -24974.151} C_VEL
LIN {X 0,Y 158.487,Z 553.282,A -85,B 0,C 180,E1 -24978.19,E2 -24978.19} C_VEL
LIN {X 0,Y 165.9,Z 541.707,A -85,B 0,C 180,E1 -24981.602,E2 -24981.602} C_VEL
LIN {X 0,Y 172.985,Z 529.755,A -85,B 0,C 180,E1 -24984.346,E2 -24984.346} C_VEL
LIN {X 0,Y 179.825,Z 516.803,A -85,B 0,C 180,E1 -24986.728,E2 -24986.728} C_VEL
LIN {X 0,Y 186.83,Z 501.784,A -85,B 0,C 180,E1 -24988.847,E2 -24988.847} C_VEL
LIN {X 0,Y 192.787,Z 486.658,A -85,B 0,C 180,E1 -24990.5,E2 -24990.5} C_VEL
LIN {X 0,Y 197.864,Z 471.214,A -85,B 0,C 180,E1 -24991.802,E2 -24991.802} C_VEL
LIN {X 0,Y 202.2,Z 454.961,A -85,B 0,C 180,E1 -24992.82,E2 -24992.82} C_VEL
LIN {X 0,Y 205.57,Z 438.624,A -85,B 0,C 180,E1 -24993.531,E2 -24993.531} C_VEL
LIN {X 0,Y 207.793,Z 421.798,A -85,B 0,C 180,E1 -24994.077,E2 -24994.077} C_VEL
LIN {X 0,Y 214.538,Z 351.325,A -85,B 0,C 180,E1 -24995.96,E2 -24995.96} C_VEL
LIN {X 0,Y 210.28,Z 341.171,A -85,B 0,C 180,E1 -24998.599,E2 -24998.599} C_VEL
LIN {X 0,Y 208.145,Z 336.806,A -85,B 0,C 180,E1 -24999.989,E2 -24999.989} C_VEL
LIN {X 0,Y 203.14,Z 327.858,A -85,B 0,C 180,E1 -25003.469,E2 -25003.469} C_VEL
LIN {X 0,Y 199.567,Z 321.852,A -85,B 0,C 180,E1 -25006.306,E2 -25006.306} C_VEL
LIN {X 0,Y 196.157,Z 316.417,A -85,B 0,C 180,E1 -25009.334,E2 -25009.334} C_VEL
LIN {X 0,Y 192.666,Z 310.719,A -85,B 0,C 180,E1 -25013.043,E2 -25013.043} C_VEL
LIN {X 0,Y 189.632,Z 306.168,A -85,B 0,C 180,E1 -25016.998,E2 -25016.998} C_VEL
LIN {X 0,Y 187.342,Z 302.66,A -85,B 0,C 180,E1 -25020.855,E2 -25020.855} C_VEL
LIN {X 0,Y 186.775,Z 301.454,A -85,B 0,C 180,E1 -25022.156,E2 -25022.156} C_VEL
LIN {X 0,Y 184.737,Z 299.224,A -85,B 0,C 180,E1 -25028.037,E2 -25028.037} C_VEL
LIN {X 0,Y 184.386,Z 297.683,A -85,B 0,C 180,E1 -25030.987,E2 -25030.987} C_VEL
LIN {X 0,Y 184.307,Z 297.486,A -85,B 0,C 180,E1 -25033.226,E2 -25033.226} C_VEL
LIN {X 0,Y 184.482,Z 299.123,A -85,B 0,C 180,E1 -25037.388,E2 -25037.388} C_VEL
LIN {X 0,Y 187.039,Z 302.463,A -85,B 0,C 180,E1 -25045.096,E2 -25045.096} C_VEL
LIN {X 0,Y 189.258,Z 306.113,A -85,B 0,C 180,E1 -25049.069,E2 -25049.069} C_VEL
LIN {X 0,Y 190.248,Z 307.505,A -85,B 0,C 180,E1 -25050.476,E2 -25050.476} C_VEL
LIN {X 0,Y 193.04,Z 311.751,A -85,B 0,C 180,E1 -25053.974,E2 -25053.974} C_VEL
LIN {X 0,Y 195.94,Z 316.241,A -85,B 0,C 180,E1 -25057.002,E2 -25057.002} C_VEL
LIN {X 0,Y 198.947,Z 321.045,A -85,B 0,C 180,E1 -25059.729,E2 -25059.729} C_VEL
LIN {X 0,Y 202.288,Z 326.434,A -85,B 0,C 180,E1 -25062.415,E2 -25062.415} C_VEL
LIN {X 0,Y 207.972,Z 336.406,A -85,B 0,C 180,E1 -25066.41,E2 -25066.41} C_VEL
LIN {X 0,Y 213.134,Z 346.21,A -85,B 0,C 180,E1 -25069.597,E2 -25069.597} C_VEL
LIN {X 0,Y 214.482,Z 348.943,A -85,B 0,C 180,E1 -25070.371,E2 -25070.371} C_VEL
LIN {X 0,Y 212.236,Z 372.631,A -85,B 0,C 180,E1 -25071.011,E2 -25071.011} C_VEL
LIN {X 0,Y 207.086,Z 424.425,A -85,B 0,C 180,E1 -25072.424,E2 -25072.424} C_VEL
LIN {X 0,Y 204.045,Z 442.308,A -85,B 0,C 180,E1 -25073.164,E2 -25073.164} C_VEL
LIN {X 0,Y 200.17,Z 458.67,A -85,B 0,C 180,E1 -25074.143,E2 -25074.143} C_VEL
LIN {X 0,Y 195.568,Z 474.04,A -85,B 0,C 180,E1 -25075.372,E2 -25075.372} C_VEL
LIN {X 0,Y 190.092,Z 489.251,A -85,B 0,C 180,E1 -25076.952,E2 -25076.952} C_VEL
LIN {X 0,Y 183.73,Z 504.107,A -85,B 0,C 180,E1 -25078.909,E2 -25078.909} C_VEL
LIN {X 0,Y 177.006,Z 517.811,A -85,B 0,C 180,E1 -25081.221,E2 -25081.221} C_VEL
LIN {X 0,Y 169.323,Z 531.457,A -85,B 0,C 180,E1 -25084.162,E2 -25084.162} C_VEL
LIN {X 0,Y 162.716,Z 542.146,A -85,B 0,C 180,E1 -25087.124,E2 -25087.124} C_VEL
LIN {X 0,Y 155.343,Z 553.101,A -85,B 0,C 180,E1 -25090.923,E2 -25090.923} C_VEL
LIN {X 0,Y 148.856,Z 562.217,A -85,B 0,C 180,E1 -25094.949,E2 -25094.949} C_VEL
LIN {X 0,Y 142.199,Z 571.152,A -85,B 0,C 180,E1 -25100.084,E2 -25100.084} C_VEL
LIN {X 0,Y 136.73,Z 578.454,A -85,B 0,C 180,E1 -25105.577,E2 -25105.577} C_VEL
LIN {X 0,Y 132.336,Z 584.529,A -85,B 0,C 180,E1 -25111.521,E2 -25111.521} C_VEL
LIN {X 0,Y 129.094,Z 589.387,A -85,B 0,C 180,E1 -25117.821,E2 -25117.821} C_VEL
LIN {X 0,Y 127.34,Z 592.27,A -85,B 0,C 180,E1 -25122.753,E2 -25122.753} C_VEL
LIN {X 0,Y 126.043,Z 595.114,A -85,B 0,C 180,E1 -25129.544,E2 -25129.544} C_VEL
LIN {X 0,Y 125.755,Z 596.869,A -85,B 0,C 180,E1 -25136.597,E2 -25136.597} C_VEL
LIN {X 0,Y 126.341,Z 597.527,A -85,B 0,C 180,E1 -25143.797,E2 -25143.797} C_VEL
LIN {X 0,Y 128.21,Z 596.934,A -85,B 0,C 180,E1 -25151.13,E2 -25151.13} C_VEL
LIN {X 0,Y 131.657,Z 595.054,A -85,B 0,C 180,E1 -25158.358,E2 -25158.358} C_VEL
LIN {X 0,Y 137.13,Z 591.596,A -85,B 0,C 180,E1 -25165.684,E2 -25165.684} C_VEL
LIN {X 0,Y 143.59,Z 587.174,A -85,B 0,C 180,E1 -25171.761,E2 -25171.761} C_VEL
LIN {X 0,Y 152.056,Z 580.987,A -85,B 0,C 180,E1 -25177.574,E2 -25177.574} C_VEL
LIN {X 0,Y 160.704,Z 574.057,A -85,B 0,C 180,E1 -25182.174,E2 -25182.174} C_VEL
LIN {X 0,Y 168.154,Z 567.569,A -85,B 0,C 180,E1 -25185.477,E2 -25185.477} C_VEL
LIN {X 0,Y 177.205,Z 559.039,A -85,B 0,C 180,E1 -25188.837,E2 -25188.837} C_VEL
LIN {X 0,Y 186.404,Z 549.37,A -85,B 0,C 180,E1 -25191.761,E2 -25191.761} C_VEL
LIN {X 0,Y 196.287,Z 537.76,A -85,B 0,C 180,E1 -25194.461,E2 -25194.461} C_VEL
LIN {X 0,Y 205.895,Z 524.971,A -85,B 0,C 180,E1 -25196.75,E2 -25196.75} C_VEL
LIN {X 0,Y 214.602,Z 511.729,A -85,B 0,C 180,E1 -25198.568,E2 -25198.568} C_VEL
LIN {X 0,Y 221.087,Z 500.283,A -85,B 0,C 180,E1 -25199.832,E2 -25199.832} C_VEL
LIN {X 0,Y 228.45,Z 485.312,A -85,B 0,C 180,E1 -25201.144,E2 -25201.144} C_VEL
LIN {X 0,Y 234.276,Z 471.243,A -85,B 0,C 180,E1 -25202.124,E2 -25202.124} C_VEL
LIN {X 0,Y 239.66,Z 455.1,A -85,B 0,C 180,E1 -25202.987,E2 -25202.987} C_VEL
LIN {X 0,Y 243.822,Z 438.822,A -85,B 0,C 180,E1 -25203.613,E2 -25203.613} C_VEL
LIN {X 0,Y 246.842,Z 422.066,A -85,B 0,C 180,E1 -25204.068,E2 -25204.068} C_VEL
LIN {X 0,Y 252.948,Z 371.872,A -85,B 0,C 180,E1 -25205.194,E2 -25205.194} C_VEL
LIN {X 0,Y 252.008,Z 368.576,A -85,B 0,C 180,E1 -25207.393,E2 -25207.393} C_VEL
LIN {X 0,Y 251.045,Z 365.288,A -85,B 0,C 180,E1 -25212.22,E2 -25212.22} C_VEL
LIN {X 0,Y 251.004,Z 365.535,A -85,B 0,C 180,E1 -25213.258,E2 -25213.258} C_VEL
LIN {X 0,Y 251.845,Z 368.791,A -85,B 0,C 180,E1 -25217.963,E2 -25217.963} C_VEL
LIN {X 0,Y 252.876,Z 371.878,A -85,B 0,C 180,E1 -25220.329,E2 -25220.329} C_VEL
LIN {X 0,Y 252.94,Z 372.463,A -85,B 0,C 180,E1 -25220.521,E2 -25220.521} C_VEL
LIN {X 0,Y 245.926,Z 429.223,A -85,B 0,C 180,E1 -25221.776,E2 -25221.776} C_VEL
LIN {X 0,Y 242.468,Z 446.09,A -85,B 0,C 180,E1 -25222.234,E2 -25222.234} C_VEL
LIN {X 0,Y 237.946,Z 462.08,A -85,B 0,C 180,E1 -25222.823,E2 -25222.823} C_VEL
LIN {X 0,Y 232.85,Z 476.467,A -85,B 0,C 180,E1 -25223.541,E2 -25223.541} C_VEL
LIN {X 0,Y 226.761,Z 490.73,A -85,B 0,C 180,E1 -25224.44,E2 -25224.44} C_VEL
LIN {X 0,Y 220.078,Z 504.005,A -85,B 0,C 180,E1 -25225.562,E2 -25225.562} C_VEL
LIN {X 0,Y 211.265,Z 518.988,A -85,B 0,C 180,E1 -25227.146,E2 -25227.146} C_VEL
LIN {X 0,Y 202.69,Z 531.665,A -85,B 0,C 180,E1 -25228.897,E2 -25228.897} C_VEL
LIN {X 0,Y 193.031,Z 544.282,A -85,B 0,C 180,E1 -25231.176,E2 -25231.176} C_VEL
LIN {X 0,Y 191.066,Z 546.579,A -85,B 0,C 180,E1 -25231.659,E2 -25231.659} C_VEL
LIN {X 0,Y 187.27,Z 550.658,A -85,B 0,C 180,E1 -25232.335,E2 -25232.335} C_VEL
LIN {X 0,Y 174.337,Z 561.908,A -85,B 0,C 180,E1 -25233.889,E2 -25233.889} C_VEL
LIN {X 0,Y 170.303,Z 565.32,A -85,B 0,C 180,E1 -25234.722,E2 -25234.722} C_VEL
LIN {X 0,Y 169.098,Z 566.423,A -85,B 0,C 180,E1 -25235.081,E2 -25235.081} C_VEL
LIN {X 0,Y 160.808,Z 573.917,A -85,B 0,C 180,E1 -25238.126,E2 -25238.126} C_VEL
LIN {X 0,Y 151.668,Z 581.466,A -85,B 0,C 180,E1 -25242.15,E2 -25242.15} C_VEL
LIN {X 0,Y 143.376,Z 587.784,A -85,B 0,C 180,E1 -25246.668,E2 -25246.668} C_VEL
LIN {X 0,Y 136.145,Z 593.039,A -85,B 0,C 180,E1 -25251.725,E2 -25251.725} C_VEL
LIN {X 0,Y 130.083,Z 597.173,A -85,B 0,C 180,E1 -25257.299,E2 -25257.299} C_VEL
LIN {X 0,Y 124.607,Z 600.856,A -85,B 0,C 180,E1 -25264.477,E2 -25264.477} C_VEL
LIN {X 0,Y 120.667,Z 603.402,A -85,B 0,C 180,E1 -25273.071,E2 -25273.071} C_VEL
LIN {X 0,Y 119.361,Z 604.22,A -85,B 0,C 180,E1 -25279.827,E2 -25279.827} C_VEL
LIN {X 0,Y 119.185,Z 604.171,A -85,B 0,C 180,E1 -25286.62,E2 -25286.62} C_VEL
LIN {X 0,Y 119.359,Z 603.74,A -85,B 0,C 180,E1 -25290.001,E2 -25290.001} C_VEL
LIN {X 0,Y 119.27,Z 603.046,A -85,B 0,C 180,E1 -25293.379,E2 -25293.379} C_VEL
LIN {X 0,Y 119.406,Z 600.942,A -85,B 0,C 180,E1 -25300.171,E2 -25300.171} C_VEL
LIN {X 0,Y 121.197,Z 596.771,A -85,B 0,C 180,E1 -25308.599,E2 -25308.599} C_VEL
LIN {X 0,Y 123.878,Z 592.377,A -85,B 0,C 180,E1 -25314.807,E2 -25314.807} C_VEL
LIN {X 0,Y 128.251,Z 586.277,A -85,B 0,C 180,E1 -25321.372,E2 -25321.372} C_VEL
LIN {X 0,Y 133.75,Z 579.16,A -85,B 0,C 180,E1 -25327.177,E2 -25327.177} C_VEL
LIN {X 0,Y 141.363,Z 569.319,A -85,B 0,C 180,E1 -25333.126,E2 -25333.126} C_VEL
LIN {X 0,Y 148.237,Z 560.11,A -85,B 0,C 180,E1 -25337.296,E2 -25337.296} C_VEL
LIN {X 0,Y 155.739,Z 549.348,A -85,B 0,C 180,E1 -25341.118,E2 -25341.118} C_VEL
LIN {X 0,Y 163.877,Z 536.677,A -85,B 0,C 180,E1 -25344.571,E2 -25344.571} C_VEL
LIN {X 0,Y 171.355,Z 523.93,A -85,B 0,C 180,E1 -25347.224,E2 -25347.224} C_VEL
LIN {X 0,Y 178.677,Z 509.791,A -85,B 0,C 180,E1 -25349.501,E2 -25349.501} C_VEL
LIN {X 0,Y 185.207,Z 495.039,A -85,B 0,C 180,E1 -25351.344,E2 -25351.344} C_VEL
LIN {X 0,Y 190.697,Z 480.457,A -85,B 0,C 180,E1 -25352.761,E2 -25352.761} C_VEL
LIN {X 0,Y 195.964,Z 463.498,A -85,B 0,C 180,E1 -25354.005,E2 -25354.005} C_VEL
LIN {X 0,Y 199.929,Z 447.351,A -85,B 0,C 180,E1 -25354.847,E2 -25354.847} C_VEL
LIN {X 0,Y 202.831,Z 431.134,A -85,B 0,C 180,E1 -25355.45,E2 -25355.45} C_VEL
LIN {X 0,Y 210.554,Z 354.237,A -85,B 0,C 180,E1 -25357.521,E2 -25357.521} C_VEL
LIN {X 0,Y 206.433,Z 344.256,A -85,B 0,C 180,E1 -25360.29,E2 -25360.29} C_VEL
LIN {X 0,Y 201.366,Z 334.768,A -85,B 0,C 180,E1 -25363.917,E2 -25363.917} C_VEL
LIN {X 0,Y 197.502,Z 328.058,A -85,B 0,C 180,E1 -25367.091,E2 -25367.091} C_VEL
LIN {X 0,Y 194.18,Z 322.545,A -85,B 0,C 180,E1 -25370.224,E2 -25370.224} C_VEL
LIN {X 0,Y 190.798,Z 317.006,A -85,B 0,C 180,E1 -25374.006,E2 -25374.006} C_VEL
LIN {X 0,Y 188.386,Z 313.059,A -85,B 0,C 180,E1 -25377.352,E2 -25377.352} C_VEL
LIN {X 0,Y 186.069,Z 309.356,A -85,B 0,C 180,E1 -25381.471,E2 -25381.471} C_VEL
LIN {X 0,Y 185.548,Z 308.352,A -85,B 0,C 180,E1 -25382.675,E2 -25382.675} C_VEL
LIN {X 0,Y 183.707,Z 306.158,A -85,B 0,C 180,E1 -25388.386,E2 -25388.386} C_VEL
LIN {X 0,Y 183.422,Z 304.781,A -85,B 0,C 180,E1 -25391.045,E2 -25391.045} C_VEL
LIN {X 0,Y 183.343,Z 304.746,A -85,B 0,C 180,E1 -25394.043,E2 -25394.043} C_VEL
LIN {X 0,Y 185.322,Z 308.755,A -85,B 0,C 180,E1 -25403.534,E2 -25403.534} C_VEL
LIN {X 0,Y 185.899,Z 309.467,A -85,B 0,C 180,E1 -25404.771,E2 -25404.771} C_VEL
LIN {X 0,Y 188.24,Z 313.262,A -85,B 0,C 180,E1 -25409.036,E2 -25409.036} C_VEL
LIN {X 0,Y 191.49,Z 318.415,A -85,B 0,C 180,E1 -25413.403,E2 -25413.403} C_VEL
LIN {X 0,Y 194.547,Z 323.351,A -85,B 0,C 180,E1 -25416.699,E2 -25416.699} C_VEL
LIN {X 0,Y 198.538,Z 329.913,A -85,B 0,C 180,E1 -25420.328,E2 -25420.328} C_VEL
LIN {X 0,Y 202.784,Z 337.439,A -85,B 0,C 180,E1 -25423.683,E2 -25423.683} C_VEL
